(* CoDeSys 2.3.9.59 project: CIP_2k.pro *)
(* Author: Damir *)
(* Libraries: My_lib.lib 13.7.21 19:36:35, SysLibTime.lib 8.11.10 13:37:48, C:\Program Files (x86)\WAGO Software\CODESYS V2.3\Targets\WAGO\Libraries\IO_IPC\Util.lib 29.6.15 10:12:14, Standard.lib, SYSLIBCALLBACK.LIB *)

(* PLC configuration (modules and I/O channels)
0750-0455 4 AI 4-20mA s.e. [Type_8_4_Channels] node 0, in %IB32 out %QB8 {INTTypePAAssignment = PLC; INTTypeModule = plugged}
  AT %IW0 [WORDOnW_I] Ch_1 Input word
  AT %IW1 [WORDOnW_I] Ch_2 Input word
  AT %IW2 [WORDOnW_I] Ch_3 Input word
  AT %IW3 [WORDOnW_I] Ch_4 Input word
0750-0455 4 AI 4-20mA s.e. [Type_8_4_Channels] node 1, in %IB32 out %QB8 {INTTypePAAssignment = PLC; INTTypeModule = plugged}
  AT %IW4 [WORDOnW_I] Ch_1 Input word
  AT %IW5 [WORDOnW_I] Ch_2 Input word
  AT %IW6 [WORDOnW_I] Ch_3 Input word
  AT %IW7 [WORDOnW_I] Ch_4 Input word
0750-0455 4 AI 4-20mA s.e. [Type_8_4_Channels] node 2, in %IB40 out %QB8 {INTTypePAAssignment = PLC; INTTypeModule = plugged}
  AT %IW8 [WORDOnW_I] Ch_1 Input word
  AT %IW9 [WORDOnW_I] Ch_2 Input word
  AT %IW10 [WORDOnW_I] Ch_3 Input word
  AT %IW11 [WORDOnW_I] Ch_4 Input word
0750-0455 4 AI 4-20mA s.e. [Type_8_4_Channels] node 3, in %IB48 out %QB8 {INTTypePAAssignment = PLC; INTTypeModule = plugged}
  AT %IW12 [WORDOnW_I] Ch_1 Input word
  AT %IW13 [WORDOnW_I] Ch_2 Input word
  AT %IW14 [WORDOnW_I] Ch_3 Input word
  AT %IW15 [WORDOnW_I] Ch_4 Input word
0750-0555 4 AO 4-20mA [Type_14_4_Channels] node 8, in %IB56 out %QB8 {INTTypePAAssignment = PLC; INTTypeModule = plugged}
  AT %QW0 [WORDOnW_Q] Ch_1 Analog output
  AT %QW1 [WORDOnW_Q] Ch_2 Analog output
  AT %QW2 [WORDOnW_Q] Ch_3 Analog output
  AT %QW3 [WORDOnW_Q] Ch_4 Analog output
0750-0555 4 AO 4-20mA [Type_14_4_Channels] node 9, in %IB64 out %QB8 {INTTypePAAssignment = PLC; INTTypeModule = plugged}
  AT %QW4 [WORDOnW_Q] Ch_1 Analog output
  AT %QW5 [WORDOnW_Q] Ch_2 Analog output
  AT %QW6 [WORDOnW_Q] Ch_3 Analog output
  AT %QW7 [WORDOnW_Q] Ch_4 Analog output
0750-1405 16 DI 24V DC 3.0ms [Type_1_16_Channels] node 11, in %IB32 out %QB16 {INTTypePAAssignment = PLC; INTTypeModule = plugged}
  AT %IX16.0 [BOOLOnX_I] Ch_1 Digital input
  AT %IX16.1 [BOOLOnX_I] Ch_2 Digital input
  AT %IX16.2 [BOOLOnX_I] Ch_3 Digital input
  AT %IX16.3 [BOOLOnX_I] Ch_4 Digital input
  AT %IX16.4 [BOOLOnX_I] Ch_5 Digital input
  AT %IX16.5 [BOOLOnX_I] Ch_6 Digital input
  AT %IX16.6 [BOOLOnX_I] Ch_7 Digital input
  AT %IX16.7 [BOOLOnX_I] Ch_8 Digital input
  AT %IX16.8 [BOOLOnX_I] Ch_9 Digital input
  AT %IX16.9 [BOOLOnX_I] Ch_10 Digital input
  AT %IX16.10 [BOOLOnX_I] Ch_11 Digital input
  AT %IX16.11 [BOOLOnX_I] Ch_12 Digital input
  AT %IX16.12 [BOOLOnX_I] Ch_13 Digital input
  AT %IX16.13 [BOOLOnX_I] Ch_14 Digital input
  AT %IX16.14 [BOOLOnX_I] Ch_15 Digital input
  AT %IX16.15 [BOOLOnX_I] Ch_16 Digital input
0750-1405 16 DI 24V DC 3.0ms [Type_1_16_Channels] node 12, in %IB32 out %QB16 {INTTypePAAssignment = PLC; INTTypeModule = plugged}
  AT %IX17.0 [BOOLOnX_I] Ch_1 Digital input
  AT %IX17.1 [BOOLOnX_I] Ch_2 Digital input
  AT %IX17.2 [BOOLOnX_I] Ch_3 Digital input
  AT %IX17.3 [BOOLOnX_I] Ch_4 Digital input
  AT %IX17.4 [BOOLOnX_I] Ch_5 Digital input
  AT %IX17.5 [BOOLOnX_I] Ch_6 Digital input
  AT %IX17.6 [BOOLOnX_I] Ch_7 Digital input
  AT %IX17.7 [BOOLOnX_I] Ch_8 Digital input
  AT %IX17.8 [BOOLOnX_I] Ch_9 Digital input
  AT %IX17.9 [BOOLOnX_I] Ch_10 Digital input
  AT %IX17.10 [BOOLOnX_I] Ch_11 Digital input
  AT %IX17.11 [BOOLOnX_I] Ch_12 Digital input
  AT %IX17.12 [BOOLOnX_I] Ch_13 Digital input
  AT %IX17.13 [BOOLOnX_I] Ch_14 Digital input
  AT %IX17.14 [BOOLOnX_I] Ch_15 Digital input
  AT %IX17.15 [BOOLOnX_I] Ch_16 Digital input
0750-1405 16 DI 24V DC 3.0ms [Type_1_16_Channels] node 13, in %IB34 out %QB16 {INTTypePAAssignment = PLC; INTTypeModule = plugged}
  AT %IX18.0 [BOOLOnX_I] Ch_1 Digital input
  AT %IX18.1 [BOOLOnX_I] Ch_2 Digital input
  AT %IX18.2 [BOOLOnX_I] Ch_3 Digital input
  AT %IX18.3 [BOOLOnX_I] Ch_4 Digital input
  AT %IX18.4 [BOOLOnX_I] Ch_5 Digital input
  AT %IX18.5 [BOOLOnX_I] Ch_6 Digital input
  AT %IX18.6 [BOOLOnX_I] Ch_7 Digital input
  AT %IX18.7 [BOOLOnX_I] Ch_8 Digital input
  AT %IX18.8 [BOOLOnX_I] Ch_9 Digital input
  AT %IX18.9 [BOOLOnX_I] Ch_10 Digital input
  AT %IX18.10 [BOOLOnX_I] Ch_11 Digital input
  AT %IX18.11 [BOOLOnX_I] Ch_12 Digital input
  AT %IX18.12 [BOOLOnX_I] Ch_13 Digital input
  AT %IX18.13 [BOOLOnX_I] Ch_14 Digital input
  AT %IX18.14 [BOOLOnX_I] Ch_15 Digital input
  AT %IX18.15 [BOOLOnX_I] Ch_16 Digital input
0750-1504 16 DO 24V DC 0.5A [Type_10_16_Channels] node 19, in %IB36 out %QB16 {INTTypePAAssignment = PLC; INTTypeModule = plugged}
  AT %QX8.0 [BOOLOnX_Q] Ch_1 Digital output
  AT %QX8.1 [BOOLOnX_Q] Ch_2 Digital output
  AT %QX8.2 [BOOLOnX_Q] Ch_3 Digital output
  AT %QX8.3 [BOOLOnX_Q] Ch_4 Digital output
  AT %QX8.4 [BOOLOnX_Q] Ch_5 Digital output
  AT %QX8.5 [BOOLOnX_Q] Ch_6 Digital output
  AT %QX8.6 [BOOLOnX_Q] Ch_7 Digital output
  AT %QX8.7 [BOOLOnX_Q] Ch_8 Digital output
  AT %QX8.8 [BOOLOnX_Q] Ch_9 Digital output
  AT %QX8.9 [BOOLOnX_Q] Ch_10 Digital output
  AT %QX8.10 [BOOLOnX_Q] Ch_11 Digital output
  AT %QX8.11 [BOOLOnX_Q] Ch_12 Digital output
  AT %QX8.12 [BOOLOnX_Q] Ch_13 Digital output
  AT %QX8.13 [BOOLOnX_Q] Ch_14 Digital output
  AT %QX8.14 [BOOLOnX_Q] Ch_15 Digital output
  AT %QX8.15 [BOOLOnX_Q] Ch_16 Digital output
0750-1504 16 DO 24V DC 0.5A [Type_10_16_Channels] node 20, in %IB38 out %QB16 {INTTypePAAssignment = PLC; INTTypeModule = plugged}
  AT %QX9.0 [BOOLOnX_Q] Ch_1 Digital output
  AT %QX9.1 [BOOLOnX_Q] Ch_2 Digital output
  AT %QX9.2 [BOOLOnX_Q] Ch_3 Digital output
  AT %QX9.3 [BOOLOnX_Q] Ch_4 Digital output
  AT %QX9.4 [BOOLOnX_Q] Ch_5 Digital output
  AT %QX9.5 [BOOLOnX_Q] Ch_6 Digital output
  AT %QX9.6 [BOOLOnX_Q] Ch_7 Digital output
  AT %QX9.7 [BOOLOnX_Q] Ch_8 Digital output
  AT %QX9.8 [BOOLOnX_Q] Ch_9 Digital output
  AT %QX9.9 [BOOLOnX_Q] Ch_10 Digital output
  AT %QX9.10 [BOOLOnX_Q] Ch_11 Digital output
  AT %QX9.11 [BOOLOnX_Q] Ch_12 Digital output
  AT %QX9.12 [BOOLOnX_Q] Ch_13 Digital output
  AT %QX9.13 [BOOLOnX_Q] Ch_14 Digital output
  AT %QX9.14 [BOOLOnX_Q] Ch_15 Digital output
  AT %QX9.15 [BOOLOnX_Q] Ch_16 Digital output
0750-1504 16 DO 24V DC 0.5A [Type_10_16_Channels] node 21, in %IB38 out %QB18 {INTTypePAAssignment = PLC; INTTypeModule = plugged}
  AT %QX10.0 [BOOLOnX_Q] Ch_1 Digital output
  AT %QX10.1 [BOOLOnX_Q] Ch_2 Digital output
  AT %QX10.2 [BOOLOnX_Q] Ch_3 Digital output
  AT %QX10.3 [BOOLOnX_Q] Ch_4 Digital output
  AT %QX10.4 [BOOLOnX_Q] Ch_5 Digital output
  AT %QX10.5 [BOOLOnX_Q] Ch_6 Digital output
  AT %QX10.6 [BOOLOnX_Q] Ch_7 Digital output
  AT %QX10.7 [BOOLOnX_Q] Ch_8 Digital output
  AT %QX10.8 [BOOLOnX_Q] Ch_9 Digital output
  AT %QX10.9 [BOOLOnX_Q] Ch_10 Digital output
  AT %QX10.10 [BOOLOnX_Q] Ch_11 Digital output
  AT %QX10.11 [BOOLOnX_Q] Ch_12 Digital output
  AT %QX10.12 [BOOLOnX_Q] Ch_13 Digital output
  AT %QX10.13 [BOOLOnX_Q] Ch_14 Digital output
  AT %QX10.14 [BOOLOnX_Q] Ch_15 Digital output
  AT %QX10.15 [BOOLOnX_Q] Ch_16 Digital output
Fieldbus variables [FB_VARS] node 1, in %IB0 out %QB0
Flag variables [FLAG_VARS] node 2, in %IB0 out %QB0
Modbus-Master [MB_MASTER] node 3, in %IB0 out %QB0
*)

(* Global variable list: Alarms *)
VAR_GLOBAL

(*----------------аварии контура 1---------------------*)
	Alarm_VA541		AT %QX256.0	: BOOL;	(*аварии клапанов*)
	Alarm_VA401    		AT %QX256.1 	: BOOL;
	Alarm_VA201    		AT %QX256.2  	: BOOL;
	Alarm_VA301    		AT %QX256.3 	: BOOL;
	Alarm_VA41     		AT %QX256.4  	: BOOL;
	Alarm_VA11     		AT %QX256.5	: BOOL;
	Alarm_VA21     		AT %QX256.6  	: BOOL;
	Alarm_VA31     		AT %QX256.7 	: BOOL;
	Alarm_VA5	    		AT %QX256.8  	: BOOL;
	Alarm_VA501    		AT %QX256.9  	: BOOL;
	Alarm_VA51     		AT %QX256.10  	: BOOL;
	Alarm_VA511    		AT %QX256.11  	: BOOL;
	Alarm_VA521    		AT %QX256.12  	: BOOL;
	Alarm_VA531    		AT %QX256.13  	: BOOL;
	Alarm_P1       		AT %QX256.14  	: BOOL;	(*авария насоса подачи*)
	Alarm_PE1        		AT %QX256.15  	: BOOL;	(*Превышение давления контур 1*)

	Alarm_FE11      		AT %QX257.0	: BOOL;	(*Нет протока на подаче контур 1*)
	AlarmBackFlow_C1 	AT %QX257.1 	: BOOL; 	(*Нет протока на возврате контур 1*)
	HeatingAlarm_C1  	AT %QX257.2 	: BOOL; 	(*Долгий нагрев контур 1*)
	CondAlarm_C1  		AT %QX257.3 	: BOOL; 	(*Долгий набор концентрации контур 1*)
	Alarm_Empty_Q5		AT %QX257.4 	: BOOL; 	(*авария опустошения цирк бака при работе на замкн маршруте*)
	Alarm_TE11      		AT %QX257.5  	: BOOL; 	(*Перегрев на выходе теплообменника контура 1*)

	Error_TE11      	AT %QX258.0 	: BOOL; (*аварии аналоговых датчиков*)
	Error_PE1        	AT %QX258.1 	: BOOL;
	Error_FE1        	AT %QX258.2  	: BOOL;
	Error_QE1        	AT %QX258.3  	: BOOL;
	Error_TE21       	AT %QX258.4  	: BOOL;


(*-----------------аварии контура 2-------------------*)
	Alarm_VA642    	AT %QX259.0  	: BOOL;
	Alarm_VA402    	AT %QX259.1  	: BOOL;
	Alarm_VA202    	AT %QX259.2 	: BOOL;
	Alarm_VA302    	AT %QX259.3 	: BOOL;
	Alarm_VA42    	AT %QX259.4  	: BOOL;
	Alarm_VA12     	AT %QX259.5  	: BOOL;
	Alarm_VA22     	AT %QX259.6 	: BOOL;
	Alarm_VA32     	AT %QX259.7 	: BOOL;
	Alarm_VA6	    	AT %QX259.8  	: BOOL;
	Alarm_VA602    	AT %QX259.9  	: BOOL;
	Alarm_VA62     	AT %QX259.10  	: BOOL;
	Alarm_VA612    	AT %QX259.11 	: BOOL;
	Alarm_VA622    	AT %QX259.12 	: BOOL;
	Alarm_VA632    	AT %QX259.13 	: BOOL;
	Alarm_P2       	AT %QX259.14  	: BOOL;	(*авария насоса подачи*)
	Alarm_PE2        	AT %QX259.15  	: BOOL; 	(*Превышение давления контур 2*)

	Alarm_FE12       		AT %QX260.0  	: BOOL;	(*Нет протока на подаче контур 2*)
	AlarmBackFlow_C2 	AT %QX260.1	: BOOL; 	(*Нет протока на возврате контур 2*)
	HeatingAlarm_C2  	AT %QX260.2  	: BOOL; 	(*Долгий нагрев контур 2*)
	CondAlarm_C2  		AT %QX260.3 	: BOOL; 	(*Долгий набор концентрации контур 2*)
	Alarm_Empty_Q6   	AT %QX260.4 	: BOOL; 	(*авария опустошения цирк бака при работе на замкн маршруте*)
	Alarm_TE12      		AT %QX260.5  	: BOOL; 	(*Перегрев на выходе теплообменника контура 2*)

	Error_TE12       	AT %QX261.0  	: BOOL;	(*аварии аналоговых датчиков*)
	Error_PE2        	AT %QX261.1 	: BOOL;
	Error_FE2        	AT %QX261.2  	: BOOL;
	Error_QE2        	AT %QX261.3  	: BOOL;
	Error_TE22       	AT %QX261.4  	: BOOL;

(*-----------------аварии контура 3-------------------*)
(*%QX262 - %QX264*)


(*------------------общие аварии---------------------*)
	Alarm_PS         		AT %QX268.0  	: BOOL; 	(*Низкое давление сжатого воздуха*)
	Alarm_Stop       		AT %QX268.1  	: BOOL; 	(*Аварийный стоп*)
	Power_loss       		AT %QX268.2  	: BOOL; 	(*подача питания на плк - перезагрузка*)
	Alarm_VA1      		AT %QX268.3  	: BOOL;		(*авария клапана подачи чистой воды в танк Q1*)
	Alarm_LS81      		AT %QX268.4  	: BOOL;		(*аварийный уровень в баке концентрата кислоты*)
	Alarm_LS82      		AT %QX268.5  	: BOOL; 	(*низкий уровень в баке концентрата кислоты*)
	Alarm_LS71      		AT %QX268.6  	: BOOL; 	(*аварийный уровень в баке концентрата щелочи*)
	Alarm_LS72      		AT %QX268.7  	: BOOL; 	(*низкий уровень в баке концентрата щелочи*)
	Alarm_LS91     		AT %QX268.8  	: BOOL; 	(*аварийный уровень в баке дезинфектанта*)
	Alarm_LS92    		AT %QX268.9  	: BOOL; 	(*низкий уровень в баке дезинфектанта*)
    	Alarm_MinLev_Q1	AT %QX268.10  	: BOOL; 	(*минимальный уровень в танке чистой воды*)
    	Alarm_MinLev_Q2 	AT %QX268.11  	: BOOL; 	(*минимальный уровень в танке щелочи*)
    	Alarm_MinLev_Q3 	AT %QX268.12  	: BOOL; 	(*минимальный уровень в танке кислоты*)


	Error_TE2        	AT %QX269.0	: BOOL;	(*аварии аналоговых датчиков*)
	Error_TE3        	AT %QX269.1  	: BOOL;
	Error_LE1        	AT %QX269.2  	: BOOL;
	Error_LE2        	AT %QX269.3  	: BOOL;
	Error_LE3        	AT %QX269.4 	: BOOL;
(*	Error_LE4        	AT %QX269.5 	: BOOL;
	Error_TE4        	AT %QX269.6  	: BOOL; *)








END_VAR

(* Global variable list: AnalogScale *)
VAR_GLOBAL
(*%QX270 - %QX362*)

(*----------------масштабированные и пересчитанные  значения-----------------------*)
(*контур 1*)
	i_TE11   				AT %QW270		: REAL;		(*температура подачи контур 1*)
	QE1         				AT %QW272 	: REAL;     	(*расчитанная концентрация % раствора контур 1*)
	i_TE21      				AT %QW274 	: REAL;    	(*температура возврата контур 1*)
	i_FE1       				AT %QW276 	: REAL;    	(*производительность подачи л/час контур 1*)
	i_PE1       				AT %QW278 	: REAL;  	(*давление подачи контура 1*)
	i_QE1       				AT %QW280 	: REAL;  	(*показание концентратомера контур 1, мСм/см*)
	QE1_priv    				AT %QW282 	: REAL;     	(*приведенная проводимость к температуре контур 1*)
	Current_VolumeFC1		AT %QW284		: REAL;		(*текуший объем расходомера дезинфектанта контур 1*)
	Current_VolumeFC11		AT %QW286		: REAL;		(*текуший объем расходомера подачи контур 1*)

(*контур 2*)
	i_TE12      				AT %QW290 	: REAL;   	(*температура подачи контур 2*)
	QE2        				AT %QW292 	: REAL;     	(*расчитанная концентрация % раствора контур 2*)
	i_TE22      				AT %QW294 	: REAL;   	(*температура возврата контур 2*)
	i_FE2       				AT %QW296 	: REAL;   	(*производительность подачи л/час контур 2*)
	i_PE2       				AT %QW298 	: REAL;  	(*давление подачи контура 2*)
	i_QE2       				AT %QW300 	: REAL;  	(*показание концентратомера контур 2, мСм/см*)
	QE2_priv    				AT %QW302 	: REAL;     	(*приведенная проводимость к температуре контур 2*)
	Current_VolumeFC2     	AT %QW304		: REAL;  	(*текуший объем расходомера дезинфектанта контур 2*)
	Current_VolumeFC12 	AT %QW306		: REAL;		(*текуший объем расходомера подачи контур 2*)

(*контур 3*)
(*%QX310 - %QX326*)


(*общие*)
	i_TE2       	AT %QW340 	: REAL;  	(*температура в танке щелочи*)
	i_TE3       	AT %QW342 	: REAL;  	(*температура в танке кислоты*)
	i_LE1       	AT %QW344 	: REAL;   	(*текущий уровень в танке чистой воды %*)
	i_LE2       	AT %QW346 	: REAL;   	(*текущий уровень в танке щелочи %*)
	i_LE3       	AT %QW348 	: REAL;   	(*текущий уровень в танке кислоты %*)
(*	i_LE4       	AT %QW350 	: REAL;   	(*текущий уровень в танке возвратной воды %*)
	i_TE4       	AT %QW352 	: REAL;  	(*температура в танке возвратной воды*) *)


END_VAR

VAR_GLOBAL RETAIN
(*структуры данных для масштабирования сигналов с аналоговых датчиков, пользовательский тип данных AnalogScale *)
(*----------------------Контур 1----------------------------------*)
	An_Scale_TE11		AT %MW0	: AnalogScale:=(Zero:=FALSE, MaxKod:=32764.0, MinKod:=0.0, MaxVal:=100.0, MinVal:=0.0, ErrorLevel:=0.01, NumbSample:=200);
	An_Scale_PE1		AT %MW20	: AnalogScale:=(Zero:=FALSE, MaxKod:=32764.0, MinKod:=0.0, MaxVal:=6.0, MinVal:=0.0, ErrorLevel:=0.01, NumbSample:=200);
	An_Scale_FE1		AT %MW40	: AnalogScale:=(Zero:=FALSE, MaxKod:=32764.0, MinKod:=0.0, MaxVal:=30000.0, MinVal:=0.0, ErrorLevel:=0.01, NumbSample:=200);
	An_Scale_QE1		AT %MW60	: AnalogScale:=(Zero:=FALSE, MaxKod:=32764.0, MinKod:=0.0, MaxVal:=500.0, MinVal:=0.0, ErrorLevel:=0.01, NumbSample:=200);
	An_Scale_TE21		AT %MW80	: AnalogScale:=(Zero:=FALSE, MaxKod:=32764.0, MinKod:=0.0, MaxVal:=100.0, MinVal:=0.0, ErrorLevel:=0.01, NumbSample:=200);

(*----------------------Контур 2----------------------------------*)
	An_Scale_TE12		AT %MW100	: AnalogScale:=(Zero:=FALSE, MaxKod:=32764.0, MinKod:=0.0, MaxVal:=100.0, MinVal:=0.0, ErrorLevel:=0.01, NumbSample:=200);
	An_Scale_PE2		AT %MW120	: AnalogScale:=(Zero:=FALSE, MaxKod:=32764.0, MinKod:=0.0, MaxVal:=6.0, MinVal:=0.0, ErrorLevel:=0.01, NumbSample:=200);
	An_Scale_FE2		AT %MW140	: AnalogScale:=(Zero:=FALSE, MaxKod:=32764.0, MinKod:=0.0, MaxVal:=30000.0, MinVal:=0.0, ErrorLevel:=0.01, NumbSample:=200);
	An_Scale_QE2		AT %MW160	: AnalogScale:=(Zero:=FALSE, MaxKod:=32764.0, MinKod:=0.0, MaxVal:=500.0, MinVal:=0.0, ErrorLevel:=0.01, NumbSample:=200);
	An_Scale_TE22		AT %MW180	: AnalogScale:=(Zero:=FALSE, MaxKod:=32764.0, MinKod:=0.0, MaxVal:=100.0, MinVal:=0.0, ErrorLevel:=0.01, NumbSample:=200);

(*----------------------общие--------------------------------*)
	An_Scale_TE2		AT %MW200	: AnalogScale:=(Zero:=FALSE, MaxKod:=32764.0, MinKod:=0.0, MaxVal:=100.0, MinVal:=0.0, ErrorLevel:=0.01, NumbSample:=200);
	An_Scale_TE3		AT %MW220	: AnalogScale:=(Zero:=FALSE, MaxKod:=32764.0, MinKod:=0.0, MaxVal:=100.0, MinVal:=0.0, ErrorLevel:=0.01, NumbSample:=200);
	An_Scale_LE1		AT %MW240	: AnalogScale:=(Zero:=FALSE, MaxKod:=32764.0, MinKod:=0.0, MaxVal:=0.25, MinVal:=0.0, ErrorLevel:=0.01, Hight_LE:=2.4, NumbSample:=200);
	An_Scale_LE2		AT %MW260	: AnalogScale:=(Zero:=FALSE, MaxKod:=32764.0, MinKod:=0.0, MaxVal:=0.25, MinVal:=0.0, ErrorLevel:=0.01, Hight_LE:=2.4, NumbSample:=200);
	An_Scale_LE3		AT %MW280	: AnalogScale:=(Zero:=FALSE, MaxKod:=32764.0, MinKod:=0.0, MaxVal:=0.25, MinVal:=0.0, ErrorLevel:=0.01, Hight_LE:=2.4, NumbSample:=200);
(*	An_Scale_LE4		AT %MW300	: AnalogScale:=(Zero:=FALSE, MaxKod:=32764.0, MinKod:=0.0, MaxVal:=0.25, MinVal:=0.0, ErrorLevel:=0.01 ,Hight_LE:=2.4, NumbSample:=200);
	An_Scale_TE4		AT %MW320	: AnalogScale:=(Zero:=FALSE, MaxKod:=32764.0, MinKod:=0.0, MaxVal:=100.0, MinVal:=0.0, ErrorLevel:=0.01, NumbSample:=200); *)



END_VAR

(* Global variable list: Constants *)
VAR_GLOBAL CONSTANT

	ar_Null_20 : ARRAY [0..20] OF BOOL := 21(FALSE) ;  (*нулевой массив для обнуления*)
	ar_Full_20 : ARRAY [0..20] OF BOOL := 21(TRUE) ;    (*заполненный массив*)

(*объявления констант для доступа к отдельным битам в словах *)
(*управление механизмами каждого контура*)
	VA541		: INT:= 0;	(*VA541 Клапан сброса в канализацию из контура *)
	VA401		: INT:= 1;	(*VA401 Клапан подачи в бак возвратной воды *)
	VA201		: INT:= 2;	(*VA201 Клапан подачи в бак щелочи *)
	VA301		: INT:= 3;	(*VA301 Клапан подачи в бак кислоты *)
	VA41		: INT:= 4;	(*VA41 Клапан выпуска из бака возвратной воды*)
	VA11		: INT:= 5;	(*VA11 Клапан выпуска из бака чистой воды*)
	VA21		: INT:= 6;	(*VA21 Клапан выпуска из бака щелочи*)
	VA31		: INT:= 7;	(*VA31 Клапан выпуска из бака кислоты*)
	VA5			: INT:= 8;	(*VA5 Клапан подачи чистой воды в цирк бак*)
	VA501		: INT:= 9;	(*VA501 Клапан подачи растворов в цирк бак*)
	VA51		: INT:= 10;	(*VA51  Клапан выпуска из цирк бака*)
	VA511		: INT:= 11;	(*VA511 Клапан выпуска в канализацию из цирк бака*)
	VA521		: INT:= 12;	(*VA521 Клапан циркуляции по контуру*)
	VA531		: INT:= 13;	(*VA531 Клапан подачи из контура в маршрут*)
	VA14		: INT:= 14;	(*VA14 Отсечной клапан пара*)
	P1			: INT:= 15;	(*Р1 Старт насоса подачи *)

	BackPump		: INT:= 16;	(*Старт насоса возврата*)
	Heating_VR1		: INT:= 17;	(*Включение нагрева*)
	VE551			: INT:= 18;	(*VE551 Клапан дезинфектанта*)
	Zero_FC11		: INT:= 19;	(*обнуление счетчика расходомера раствора, в ручном режиме*)
	Zero_FC1		: INT:= 20;	(*обнуление счетчика расходомера дезинфектанта, в ручном режиме*)


END_VAR

(* Global variable list: DeviceControl *)
VAR_GLOBAL

(*-------------состояние механизмов с диагностикой контур 1-------------*)
	Mode_VA541 	AT %QW360: INT;
	Mode_VA401    	AT %QW361: INT;
	Mode_VA201    	AT %QW362: INT;
	Mode_VA301    	AT %QW363: INT;
	Mode_VA41     	AT %QW364: INT;
	Mode_VA11     	AT %QW365: INT;
	Mode_VA21     	AT %QW366: INT;
	Mode_VA31     	AT %QW367: INT;
	Mode_VA5    	AT %QW368: INT;
	Mode_VA501    	AT %QW369: INT;
	Mode_VA51     	AT %QW370: INT;
	Mode_VA511    	AT %QW371: INT;
	Mode_VA521    	AT %QW372: INT;
	Mode_VA531    	AT %QW373: INT;
	Mode_P1     		AT %QW374: INT;


(*-------------состояние  механизмов с диагностикой контур 2-------------*)
	Mode_VA642    	AT %QW380: INT;
	Mode_VA402    	AT %QW381: INT;
	Mode_VA202    	AT %QW382: INT;
	Mode_VA302    	AT %QW383: INT;
	Mode_VA42    	AT %QW384: INT;
	Mode_VA12     	AT %QW385: INT;
	Mode_VA22     	AT %QW386: INT;
	Mode_VA32     	AT %QW387: INT;
	Mode_VA6    	AT %QW388: INT;
	Mode_VA602    	AT %QW389: INT;
	Mode_VA62     	AT %QW390: INT;
	Mode_VA612    	AT %QW391: INT;
	Mode_VA622    	AT %QW392: INT;
	Mode_VA632    	AT %QW393: INT;
	Mode_P2     		AT %QW394: INT;

(*-------------состояние механизмов с диагностикой контур 3-------------*)
(*%QW400 - %QW414*)


(*------------состояние общих механизмов с диагностикой--------------*)
	Mode_VA1      	AT %QW439: INT;

(*------------------------------------------------------------------------------------------*)

(*------------------команды управления механизмами------------------*)
(*контур 1*)
	w_qDevice_C1		AT%QW440	:DWORD; 	(*слово команд управления механизмами контура 1*)
	q_P1an  			AT%QW442 	: REAL;		(*аналоговое задание на насос подачи*)
	q_VR1an 			AT%QW444 	: REAL;		(*аналоговое задание на регулирующий клапан пара*)
	SP_VR1							: REAL;		(*задание температуры на регулятор*)
	SP_P1  							: REAL;	 	(*задание производительности на регулятор*)

(*контур 2*)
	w_qDevice_C2		AT%QW446	:DWORD; 	(*слово команд управления механизмами контура 2*)
	q_P2an  			AT%QW448 	: REAL;
	q_VR2an 			AT%QW450 	: REAL;
	SP_VR2 						: REAL;	 	(*задание температуры на регулятор*)
	SP_P2  							: REAL;	 	(*задание производительности на регулятор*)

(*контур 3*)
(*%QW452 - %QW458*)

(*общие механизмы*)
	q_VA1      			AT %QX462.0	: BOOL;		(*VA1  Клапан подачи в бак чистой воды*)
	q_VE7     			AT %QX462.1	: BOOL;		(*VE7 Клапан промывки линии концентрата щелочи*)
	q_P8     				AT %QX462.2	: BOOL;		(*Р8 Насос-дозатор концентрата  кислоты*)
	q_P9     				AT %QX462.3	: BOOL;		(*Р9 Насос-дозатор концентрата  щелочи*)
	q_P10     			AT %QX462.4	: BOOL;		(*Р10 Насос-дозатор дезинфектанта*)

(*----------------------------------------------------------------------------------*)





END_VAR

VAR_GLOBAL RETAIN
(*вкл/выкл контроля положения клапанов*)
	wDiagVA_C1		AT%MW400		:WORD:= 16#FF ;	(*контроль состояния клапанов с диагностикой контур 1*)
	wDiagVA_C2		AT%MW401		:WORD:= 16#FF;	(*контроль состояния клапанов с диагностикой контур 2*)
	DiagVA1      			AT %MX402.0  	: BOOL:= TRUE;		(*контроль состояния клапана подачи в танк чистой воды*)

(*--------настройки ПИД-регуляторов-------------*)
(*контур 1*)
	SP_PID_P_VR1		AT %MW404	: REAL := 1.3;     	(*коеф усиления ПИД р-ра температуры*)
	SP_PID_I_VR1   	AT %MW406	: REAL := 10.0;    	(*время интегрирования ПИД р-ра температуры *)
	SP_PID_P_P1    	AT %MW408	: REAL := 0.5;     	(*коеф усиления ПИД р-ра расхода*)
	SP_PID_I_P1     		AT %MW410	: REAL := 10.0;    	(*время интегрирования ПИД р-ра расхода *)

(*контур 2*)
	SP_PID_P_VR2		AT %MW412	: REAL := 1.3;     	(*коеф усиления ПИД р-ра температуры*)
	SP_PID_I_VR2 		AT %MW414	: REAL := 10.0; 		(*время интегрирования ПИД р-ра температуры *)
	SP_PID_P_P2   		AT %MW416	: REAL := 0.3;     	(*коеф усиления ПИД р-ра расхода*)
	SP_PID_I_P2    		AT %MW418	: REAL := 10.0;    	(*время интегрирования ПИД р-ра расхода *)

(*------------вес импульса расходомера--------------*)
(*контур 1*)
	K_imp_C1         		AT %MW438	: REAL := 0.1;    		(*литр/имп расходомера подачи*)
	K_imp_dez_C1 		AT %MW440	: REAL := 5.0;     	(*мл/имп расходомера дезинфектанта*)
(*контур 2*)
	K_imp_C2        		AT %MW442	: REAL := 0.1;		(*литр/имп расходомера подачи*)
	K_imp_dez_C2 		AT %MW444	: REAL := 5.0;		(*мл/имп расходомера дезинфектанта*)


END_VAR

(* Global variable list: Global_Variables *)
VAR_GLOBAL
	scan_time : REAL;    (*время скана, из fb_TimeIncr*)


END_VAR

VAR_GLOBAL RETAIN

	Mode_Q1               	AT %MW500	: INT;  		(*режим пополнения бака Q1 чистой воды*)
	MaxLevel_Q1           	AT %MW501	: INT := 90;	(*макс уровень в танке чистой воды - поддержание уровня,%*)
	MinLevel_Q1          	AT %MW502	: INT := 70;  	(*мин уровень в танке чистой воды - поддержание уровня,%*)

	MinAlarmLevel_Q1   	AT %MW503	: INT := 20; 	(*мин уровень в танке чистой воды Q1,%*)
	MinAlarmLevel_Q2   	AT %MW504	: INT := 20;  	(*мин уровень в танке щелочи Q2,%*)
	MinAlarmLevel_Q3  	AT %MW505	: INT := 20;  	(*мин уровень в танке кислоты Q3,%*)
	MinAlarmLevel_Q4  	AT %MW506	: INT := 20;  	(*мин уровень в танке возврат воды Q4,%*)

	Time_LSH_on          	AT %MW508	: DINT := 1;		(*время задержки датчика верхнего уровня в цирк баке,сек*)
	Time_LSM_on         	AT %MW510	: DINT := 3; 		(*время задержки датчика среднего уровня в цирк баке,сек*)
	Time_LSM_off       	AT %MW512	: DINT := 2; 		(*время задержки датчика среднего уровня в цирк баке,сек*)
	Time_LSL_off       	AT %MW514	: DINT := 2; 		(*время задержки датчика нижнего уровня в цирк баке,сек*)

	Time_Control_TE    	AT %MW516	: DINT := 7; 		(*контрольное время набора температуры, мин*)
	Time_Control_QE    	AT %MW518	: DINT := 10;		(*контрольное время набора концентрации, мин*)
	Time_Alarm_FE       	AT %MW520	: DINT := 18;		(*время аварии протока на подаче, сек*)

	MaxPressure_C1   	AT %MW524	: REAL := 4.3;     (*уставка аварии по давлению контур 1*)
	MaxPressure_C2    	AT %MW526	: REAL := 4.3;     (*уставка аварии по давлению контур 2*)

	TimeDelay_C1       	AT %MW528	: DINT := 2;       	(*время задержки вкл/выкл клапанов и насосов контур 1*)
	TimeDelay_C2      	AT %MW530	: DINT := 2;       	(*время задержки вкл/выкл клапанов и насосов контур 2*)








END_VAR

(* Global variable list: HandMode *)
VAR_GLOBAL

    (*контур 1*)
	w_ManDevice_C1	AT%MW600	:DWORD; 	(*слово команд ручного режима контура 1*)
	ManSP_P1        		AT%MW602 : REAL;		(*задание производительности насоса подачи в ручном режиме*)
	ManSP_VR1       	AT%MW604 : REAL;		(*задание температуры нагрева в ручном режиме*)


    (*контур 2*)
	w_ManDevice_C2	AT%MW606	:DWORD; 	(*слово команд ручного режима контура 2*)
	ManSP_P2        		AT%MW608 : REAL;		(*задание производительности насоса подачи в ручном режиме*)
	ManSP_VR2       	AT%MW610 : REAL;		(*задание температуры нагрева в ручном режиме*)


    (*общие механизмы*)
	Man_VA1        	AT %MX626.0 	: BOOL;		(*VA1  Клапан подачи в бак чистой воды*)
	Man_VE7        	AT %MX626.1 	: BOOL;		(*VE7 Клапан промывки линии концентрата щелочи*)
	Man_P8          	AT %MX626.2 	: BOOL;		(*Р8 Насос-дозатор концентрата  кислоты*)
	Man_P9         	AT %MX626.3	: BOOL;		(*Р9 Насос-дозатор концентрата  щелочи*)
	Man_P10         	AT %MX626.4	: BOOL;		(*Р10 Насос-дозатор дезинфектанта*)

END_VAR

(* Global variable list: Inputs *)
VAR_GLOBAL
(*---------------переменные привязанные к физическим входам----------------------------*)

(*аналоговые входа*)
	TE11_i 	AT %IW0:  WORD;	(*ТЕ11 Температура на выходе нагревателя контур 1*)
	TE12_i 	AT %IW1:  WORD;	(*ТЕ12 Температура на выходе нагревателя контур 2*)
	TE2_i   	AT %IW2:  WORD;	(*ТЕ2 Температура в танке раствора щелочи Q2*)
	TE3_i	AT %IW3:  WORD;	(*ТЕ3 Температура в танке раствора кислоты Q3*)

	LE1_i  	AT %IW4:  WORD;	(*LE1 Датчик уровня в баке чистой воды*)
	LE2_i  	AT %IW5:  WORD;	(*LE2 Датчик уровня в баке щелочи*)
	LE3_i  	AT %IW6:  WORD;	(*LE3 Датчик уровня в баке кислоты*)
	PE1_i  	AT %IW7:  WORD;	(*PE1 Датчик давления контур 1*)

	PE2_i  	AT %IW8:  WORD;	(*PE2 Датчик давления контур 2*)
	FE1_i  	AT %IW9:  WORD;	(*Производительность подачи контур 1*)
	FE2_i 	AT %IW10: WORD;	(*Производительность подачи контур 2*)
(*	    		AT %IW11: WORD;	резерв*)

	QE1_i  	AT %IW12: WORD;	(*QE1 Проводимость контур 1*)
	TE21_i 	AT %IW13: WORD;	(*TE21 Температура на возврате контур 1*)
	QE2_i   	AT %IW14: WORD;	(*QE2 Проводимость контур 2*)
	TE22_i 	AT %IW15: WORD;	(*TE22 Температура на возврате контур 2*)

(*дискретные входа*)
	VA541_i		AT %IX16.0:  BOOL; 	(*датчик положения клапана*)
	VA642_i   	AT %IX16.1:  BOOL;	(*датчик положения клапана*)
	VA401_i    	AT %IX16.2:  BOOL;	(*датчик положения клапана*)
	VA402_i    	AT %IX16.3:  BOOL;	(*датчик положения клапана*)
	VA1_i         	AT %IX16.4:  BOOL;	(*датчик положения клапана*)
	VA201_i      	AT %IX16.5:  BOOL;	(*датчик положения клапана*)
	VA202_i      	AT %IX16.6:  BOOL;	(*датчик положения клапана*)
	VA301_i     	AT %IX16.7:  BOOL;	(*датчик положения клапана*)
	VA302_i     	AT %IX16.8:  BOOL;	(*датчик положения клапана*)
	VA41_i     	AT %IX16.9:  BOOL;	(*датчик положения клапана*)
	VA42_i      	AT %IX16.10: BOOL;	(*датчик положения клапана*)
	VA11_i      	AT %IX16.11: BOOL;	(*датчик положения клапана*)
	VA12_i     	AT %IX16.12: BOOL;	(*датчик положения клапана*)
	VA21_i     	AT %IX16.13: BOOL;	(*датчик положения клапана*)
	VA22_i     	AT %IX16.14: BOOL;	(*датчик положения клапана*)
	VA31_i     	AT %IX16.15: BOOL;	(*датчик положения клапана*)

	VA32_i      	AT %IX17.0:  BOOL;	(*датчик положения клапана*)
	VA5_i       	AT %IX17.1:  BOOL;	(*датчик положения клапана*)
	VA501_i      	AT %IX17.2:  BOOL;	(*датчик положения клапана*)
	VA51_i     	AT %IX17.3:  BOOL;	(*датчик положения клапана*)
	VA511_i      	AT %IX17.4:  BOOL;	(*датчик положения клапана*)
	FS21_i      	AT %IX17.5:  BOOL;	(*FS21 Датчик протока на возврате контура 1*)
	VA521_i     	AT %IX17.6:  BOOL;	(*датчик положения клапана*)
	VA531_i     	AT %IX17.7:  BOOL;	(*датчик положения клапана*)
	LSL5_i      	AT %IX17.8:  BOOL;	(*LSL5 Датчик нижнего уровня в цирк баке Q5*)
	LSM5_i     	AT %IX17.9:  BOOL;	(*LSM5 Датчик среднего уровня в цирк баке Q5*)
	LSH5_i      	AT %IX17.10: BOOL;	(*LSH5 Датчик верхнего уровня в цирк баке Q5*)
	VA6_i        	AT %IX17.11: BOOL;	(*датчик положения клапана*)
	VA602_i   	AT %IX17.12: BOOL;	(*датчик положения клапана*)
	VA62_i       	AT %IX17.13: BOOL;	(*датчик положения клапана*)
	VA612_i      	AT %IX17.14: BOOL;	(*датчик положения клапана*)
	FS22_i      	AT %IX17.15: BOOL;	(*FS22 Датчик протока на возврате контура 2*)


	VA622_i      	AT %IX18.0:  BOOL;	(*датчик положения клапана*)
	VA632_i      	AT %IX18.1:  BOOL;	(*датчик положения клапана*)
	LSL6_i       	AT %IX18.2:  BOOL;	(*LSL6 Датчик нижнего уровня в цирк баке Q6*)
	LSM6_i       	AT %IX18.3:  BOOL;	(*LSM6 Датчик среднего уровня в цирк баке Q6*)
	LSH6_i      	AT %IX18.4:  BOOL;	(*LSH6 Датчик верхнего уровня в цирк баке Q6*)
	LS71_i    	AT %IX18.5:  BOOL;	(*LS71 Датчик аварийного нижнего уровня в баке концентрата щелочи Q7*)
	LS72_i       	AT %IX18.6:  BOOL;	(*LS72 Датчик нижнего уровня в баке концентрата щелочи Q7*)
	LS81_i      	AT %IX18.7:  BOOL;	(*LS81 Датчик аварийного нижнего уровня в баке концентрата кислоты Q8*)
	LS82_i      	AT %IX18.8:  BOOL;	(*LS82 Датчик нижнего уровня в баке концентрата кислоты Q8*)
	PS1_i      	AT %IX18.9:  BOOL;	(*PS1 Датчик давления сжатого воздуха*)
	FC1_i       	AT %IX18.10: BOOL;	(*Расход раствора контур 1, имп*)
	FC2_i       	AT %IX18.11: BOOL;	(*Расход раствора контур 2, имп*)
	ProtectP1_i 	AT %IX18.12: BOOL;	(*Готовность частоного преобразователя насоса М1*)
	ProtectP2_i 	AT %IX18.13: BOOL;	(*Готовность частоного преобразователя насоса М2*)
	AlarmStop_i	AT %IX18.14: BOOL;	(*SB1 Аварийная стоповая кнопка пульта управления*)
(*	       		AT %IX18.15: BOOL;  резерв*)




END_VAR

(* Global variable list: OP_Comands *)
VAR_GLOBAL

	AlarmReset      					AT %MX700.0: BOOL; 	(*Сброс ошибок*)

END_VAR

(* Global variable list: Outputs *)
VAR_GLOBAL
(*переменные привязанные к физическим выходам*)
(*аналоговые выходы*)
	VR1an_q   	AT %QW0 : WORD;		(*VR1 Регулирующий клапан пара контур 1*)
	VR2an_q   	AT %QW1 : WORD;		(*VR2 Регулирующий клапан пара контур 2*)
(*   				AT %QW2 : WORD;
			   	AT %QW3 : WORD;  *)

	P1an_q    	AT %QW4 : WORD;		(*Задание скорости насоса подачи контура 1*)
	P2an_q    	AT %QW5 : WORD;		(*Задание скорости насоса подачи контура 2*)
(*			    	AT %QW6 : WORD;
			    	AT %QW7 : WORD;  *)


(*дискретные выходы*)
	q_Red    	AT %QX8.0  	: BOOL;		(*Светозвуковая сигнализация. Красный свет*)
	q_Yellow   	AT %QX8.1  	: BOOL;		(*Светозвуковая сигнализация. Желтый свет*)
	q_Green   	AT %QX8.2  	: BOOL;		(*Светозвуковая сигнализация. Зеленый свет*)
	q_Sirena   	AT %QX8.3  	: BOOL;		(*Светозвуковая сигнализация. Зуммер*)
	VE7_q   	AT %QX8.4  	: BOOL;		(*VE7 Клапан промывки линии концентрата щелочи*)
	P1_q     	AT %QX8.5  	: BOOL;		(*Старт частотного преобразователя насоса М1 контура 1*)
	P2_q   		AT %QX8.6  	: BOOL;		(*Старт частотного преобразователя насоса М2 контура 2*)
	H1_q   		AT %QX8.7  	: BOOL;		(*Насос возврата Н1*)
	H2_q   		AT %QX8.8  	: BOOL;		(*Насос возврата Н2*)
	H3_q   		AT %QX8.9  	: BOOL;		(*Насос возврата Н3*)
	H4_q   		AT %QX8.10	: BOOL;		(*Насос возврата Н4*)
	H5_q   		AT %QX8.11	: BOOL;		(*Насос возврата Н5*)
	H6_q   		AT %QX8.12	: BOOL;		(*Насос возврата Н6*)
	H7_q   		AT %QX8.13	: BOOL;		(*Насос возврата Н7*)
	H8_q   		AT %QX8.14	: BOOL;		(*Насос возврата Н8*)
	H9_q   		AT %QX8.15	: BOOL;		(*Насос возврата Н9*)

	VA541_q   	AT %QX9.0  	: BOOL;		(*VA541 Клапан сброса в канализацию из контура 1*)
	VA642_q   	AT %QX9.1  	: BOOL;		(*VA642 Клапан сброса в канализацию из контура 2*)
	VA1_q    	AT %QX9.2  	: BOOL;		(*VA1  Клапан подачи в бак чистой воды*)
	VA201_q    	AT %QX9.3  	: BOOL;		(*VA201 Клапан подачи в бак щелочи контур 1*)
	VA202_q    	AT %QX9.4  	: BOOL;		(*VA202 Клапан подачи в бак щелочи контур 2*)
	VA301_q    	AT %QX9.5  	: BOOL;		(*VA301 Клапан подачи в бак кислоты контур 1*)
	VA302_q    	AT %QX9.6  	: BOOL;		(*VA302 Клапан подачи в бак кислоты контур 2*)
	VA11_q    	AT %QX9.7  	: BOOL;		(*VA11 Клапан выпуска из бака чистой воды контур 1*)
	VA12_q    	AT %QX9.8  	: BOOL;		(*VA12 Клапан выпуска из бака чистой воды контур 2*)
	VA21_q    	AT %QX9.9  	: BOOL;		(*VA21 Клапан выпуска из бака щелочи контур 1*)
	VA22_q    	AT %QX9.10	: BOOL;		(*VA22 Клапан выпуска из бака щелочи контур 2*)
	VA31_q    	AT %QX9.11	: BOOL;		(*VA31 Клапан выпуска из бака кислоты контур 1*)
	VA32_q    	AT %QX9.12	: BOOL;		(*VA32 Клапан выпуска из бака кислоты контур 2*)
	VA5_q    	AT %QX9.13	: BOOL;		(*VA5 Клапан подачи чистой воды в цирк бак контур 1*)
	VA501_q    	AT %QX9.14	: BOOL;		(*VA501 Клапан подачи растворов в цирк бак контур 1*)
	VA51_q    	AT %QX9.15	: BOOL;		(*VA51  Клапан выпуска из цирк бака контур 1*)

	VA511_q    	AT %QX10.0	: BOOL;		(*VA511 Клапан выпуска в канализацию из цирк бака контур 1*)
	VA521_q    	AT %QX10.1	: BOOL;		(*VA521 Клапан циркуляции по контуру 1*)
	VA531_q   	AT %QX10.2	: BOOL;		(*VA531 Клапан подачи из контура 1*)
	VA14_q   	AT %QX10.3	: BOOL;		(*VA14 Отсечной клапан пара контур 1*)
	VA6_q    	AT %QX10.4	: BOOL;		(*VA6 Клапан подачи чистой воды в цирк бак контур 2*)
	VA602_q   	AT %QX10.5	: BOOL;		(*VA602 Клапан подачи растворов в цирк бак контур 2*)
	VA62_q   	AT %QX10.6	: BOOL;		(*VA62  Клапан выпуска из цирк бака контур 2*)
	VA612_q   	AT %QX10.7	: BOOL;		(*VA612 Клапан выпуска в канализацию из цирк бака контур 2*)
	VA622_q    	AT %QX10.8	: BOOL;		(*VA622 Клапан циркуляции по контуру 2*)
	VA632_q   	AT %QX10.9	: BOOL;		(*VA632 Клапан подачи из контура 2*)
	VA24_q   	AT %QX10.10: BOOL;			(*VA24 Отсечной клапан пара контур 2*)
	P8_q    		AT %QX10.11: BOOL;			(*Р8 Насос-дозатор концентрата  кислоты*)
	P9_q   		AT %QX10.12: BOOL;			(*Р9 Насос-дозатор концентрата  щелочи*)
(*	   			AT %QX10.13: BOOL;
	   			AT %QX10.14: BOOL;
	    			AT %QX10.15: BOOL; *)

END_VAR

(* Global variable list: Process_Settings *)
VAR_GLOBAL RETAIN

(*----------Контур 1---------------------*)
	AlkMixing_C1           			AT %MX800.0: BOOL;     		(*перемешивание щелочи*)
	AcidMixing_C1          			AT %MX800.1: BOOL;          	(*перемешивание кислоты*)

	Stop_C1                     		AT %MX801.0 : BOOL; 		(*принудительная остановка процесса*)
	Start_AutoWashing_C1        	AT %MX801.1 : BOOL; 		(*старт мойки в автомате*)
	Start_HandMode_C1           	AT %MX801.2 : BOOL; 		(*старт ручного режима*)
	Start_PrepareAlkaline_C1   	AT %MX801.3 : BOOL; 		(*старт подготовки раствора щелочи*)
	Start_PrepareAcid_C1        	AT %MX801.4 : BOOL; 		(*старт подготовки раствора кислоты*)
	Start_Diagnostic_C1         	AT %MX801.5 : BOOL; 		(*старт диагностики клапанов*)
	ch_SwillBackWater_C1        	AT %MX801.6 : BOOL:= FALSE; 		(*выбор операции мойки*)
	ch_SwillFreshWater_C1       	AT %MX801.7 : BOOL; 		(*выбор операции мойки*)
	ch_WashAlkaline_C1          	AT %MX801.8 : BOOL; 		(*выбор операции мойки*)
	ch_WashWater1_C1            	AT %MX801.9 : BOOL; 		(*выбор операции мойки*)
	ch_WashAcid_C1              	AT %MX801.10: BOOL;		(*выбор операции мойки*)
	ch_WashWater2_C1            	AT %MX801.11: BOOL; 		(*выбор операции мойки*)
	ch_ThermDesinfection_C1 	AT %MX801.12: BOOL; 		(*выбор операции мойки*)
	ch_ChemicDesinfection_C1	AT %MX801.13: BOOL:= FALSE; 		(*выбор операции мойки*)
	Pause_C1                    		AT %MX801.14: BOOL; 		(*пауза процесса*)


	TimeSwillBackWater_C1  		AT %MW810: DINT := 300;    	(*время полоскания возвратной водой,с*)
	TimeSwillFreshWater_C1 		AT %MW812: DINT := 300;   	(*время полоскания свежей водой,с*)
	TimeWashWater1_C1      		AT %MW814: DINT := 4;       	(*время мойки 1 чистой водой,мин*)
	TempWashWater1_C1      	AT %MW816: REAL := 40.0;  	(*температруа мойки 1 чистой водой*)
	TimeWashWater2_C1      		AT %MW818: DINT := 5;       	(*время мойки 2 чистой водой,мин*)
	TempWashWater2_C1      	AT %MW820: REAL := 40.0;  	(*температруа мойки 2 чистой водой*)
	TimeWashAlkaline_C1    		AT %MW822: DINT := 20;    	(*время мойки щелочью,мин*)
	TempWashAlkaline_C1    		AT %MW824: REAL := 75.0;  	(*температура мойки щелочью*)
	TimeAlkalineMix_C1     		AT %MW826: DINT := 60;     	(*время перемешивания при мойке щелочью,с*)
	TimeWashAcid_C1        		AT %MW828: DINT := 20;     	(*время мойки кислотой,мин*)
	TempWashAcid_C1        		AT %MW830: REAL := 65.0;  	(*температура мойки кислотой*)
	TimeAcidMix_C1         		AT %MW832: DINT := 60;     	(*время перемешивания при мойке кислотой,c*)
	TimeThermDesinf_C1     		AT %MW834: DINT := 10;     	(*время термической дезинфекции,мин*)
	TempThermDesinf_C1     		AT %MW836: REAL := 85.0;  	(*температура термической дезинфекции*)
	TempCoolThermDesinf_C1 	AT %MW838: REAL := 15.0;  	(*температура охлаждения терм дезинфекции*)
	TimeChemicDesinf_C1    		AT %MW840: DINT := 10;     	(*время химической дезинфекции,мин*)
	TimeSwillChemic_C1     		AT %MW842: DINT := 15;   	(*время ополаскивания чистой водой после хим дезинфекции*)
	TimeSwillWashWater1_C1    	AT %MW844: DINT := 5;  	(*время промывки водой со сбросом в Q4 после мойки 1 чистой водой,мин*)
	TimeSwillWashWater2_C1    	AT %MW846: DINT := 5;  	(*время промывки водой со сбросом в Q4 после мойки 2 чистой водой,мин*)

	(*рецепт*)
	RouteType_C1           		AT %MW870: DINT ;           	(*тип маршрута 1 - емкостной, 0 - замкнутый*)
	PumpCapacity_C1        		AT %MW872: DINT ;           	(*производительность подающего насоса *)
	TimeDelayRetPump_C1    	AT %MW874: DINT ;           	(*время задержки включения насоса возврата*)
	TimeDelayRetFlow_C1    		AT %MW876: DINT ;           	(*время появления протока на возврате*)
	TimeAlarmBackFlow_C1   		AT %MW878: DINT ;           	(*время аварии отсутствия обратного протока*)
	Numb_BackPump_C1       	AT %MW880: DINT ;           	(*номер насоса возврата*)
	VolumeDesinf_C1        		AT %MW882: DINT ;           	(*объем дезинфектанта*)
	Using_Q5_C1             		AT %MW884: DINT ;           	(*использование циркуляционного бака на мойках растворами и водой, 1 - использовать*)
	DeltaTempStartTime_C1  		AT %MW886: DINT ;           	(*перепад температуры TE1-TE2 для начала терм дезинфекции*)
	Route_C1               			AT %MW888: DINT ;           	(*номер выбранного маршрут контура*)


(*----------Контур 2---------------------*)
	AlkMixing_C2           			AT %MX900.0: BOOL;         	(*перемешивание щелочи*)
	AcidMixing_C2          			AT %MX900.1: BOOL;          	(*перемешивание кислоты*)

	Stop_C2                     		AT %MX901.0 : BOOL; 		(*принудительная остановка процесса*)
	Start_AutoWashing_C2        	AT %MX901.1 : BOOL; 		(*старт мойки в автомате*)
	Start_HandMode_C2           	AT %MX901.2 : BOOL; 		(*старт ручного режима*)
	Start_PrepareAlkaline_C2   	AT %MX901.3 : BOOL; 		(*старт подготовки раствора щелочи*)
	Start_PrepareAcid_C2        	AT %MX901.4 : BOOL; 		(*старт подготовки раствора кислоты*)
	Start_Diagnostic_C2         	AT %MX901.5 : BOOL; 		(*старт диагностики клапанов*)
	ch_SwillBackWater_C2        	AT %MX901.6 : BOOL:= FALSE; 		(*выбор операции мойки*)
	ch_SwillFreshWater_C2       	AT %MX901.7 : BOOL; 		(*выбор операции мойки*)
	ch_WashAlkaline_C2          	AT %MX901.8 : BOOL; 		(*выбор операции мойки*)
	ch_WashWater1_C2            	AT %MX901.9 : BOOL; 		(*выбор операции мойки*)
	ch_WashAcid_C2              	AT %MX901.10 : BOOL;		(*выбор операции мойки*)
	ch_WashWater2_C2            	AT %MX901.11: BOOL; 		(*выбор операции мойки*)
	ch_ThermDesinfection_C2  	AT %MX901.12: BOOL; 		(*выбор операции мойки*)
	ch_ChemicDesinfection_C2  	AT %MX901.13: BOOL:= FALSE; 		(*выбор операции мойки*)
	Pause_C2                    		AT %MX901.14: BOOL; 		(*пауза процесса*)


	TimeSwillBackWater_C2  		AT %MW910: DINT := 300;    	(*время полоскания возвратной водой,с*)
	TimeSwillFreshWater_C2 		AT %MW912: DINT := 300;    	(*время полоскания свежей водой,с*)
	TimeWashWater1_C2      		AT %MW914: DINT := 4;       	(*время мойки 1 чистой водой,мин*)
	TempWashWater1_C2      	AT %MW916: REAL := 40.0;  	(*температруа мойки 1 чистой водой*)
	TimeWashWater2_C2      		AT %MW918: DINT := 4;       	(*время мойки 2 чистой водой,мин*)
	TempWashWater2_C2      	AT %MW920: REAL := 40.0;  	(*температруа мойки 2 чистой водой*)
	TimeWashAlkaline_C2    		AT %MW922: DINT := 30;     	(*время мойки щелочью,мин*)
	TempWashAlkaline_C2    		AT %MW924: REAL := 75.0;  	(*температура мойки щелочью*)
	TimeAlkalineMix_C2     		AT %MW926: DINT := 60;     	(*время перемешивания при мойке щелочью,с*)
	TimeWashAcid_C2        		AT %MW928: DINT := 30;     	(*время мойки кислотой,мин*)
	TempWashAcid_C2        		AT %MW930: REAL := 65.0;  	(*температура мойки кислотой*)
	TimeAcidMix_C2         		AT %MW932: DINT := 60;     	(*время перемешивания при мойке кислотой,c*)
	TimeThermDesinf_C2     		AT %MW934: DINT := 10;      	(*время термической дезинфекции,мин*)
	TempThermDesinf_C2     		AT %MW936: REAL := 85.0;  	(*температура термической дезинфекции*)
	TempCoolThermDesinf_C2 	AT %MW938: REAL := 15.0;  	(*температура охлаждения терм дезинфекции*)
	TimeChemicDesinf_C2    		AT %MW940: DINT := 10;     	(*время химической дезинфекции,мин*)
	TimeSwillChemic_C2     		AT %MW942: DINT := 15;    	(*время ополаскивания чистой водой после хим дезинфекции*)
	TimeSwillWashWater1_C2    	AT %MW944: DINT := 5;  	(*время промывки водой со сбросом в Q4 после мойки 1 чистой водой,мин*)
	TimeSwillWashWater2_C2    	AT %MW946: DINT := 5;  	(*время промывки водой со сбросом в Q4 после мойки 2 чистой водой,мин*)

	(*рецепт*)
	RouteType_C2           		AT %MW970: DINT ;           	(*тип маршрута 1 - емкостной, 0 - замкнутый*)
	PumpCapacity_C2        		AT %MW972: DINT ;           	(*производительность подающего насоса *)
	TimeDelayRetPump_C2    	AT %MW974: DINT ;           	(*время задержки включения насоса возврата*)
	TimeDelayRetFlow_C2    		AT %MW976: DINT ;           	(*время появления протока на возврате*)
	TimeAlarmBackFlow_C2   		AT %MW978: DINT ;           	(*время аварии отсутствия обратного протока*)
	Numb_BackPump_C2       	AT %MW980: DINT ;           	(*номер насоса возврата*)
	VolumeDesinf_C2        		AT %MW982: DINT ;           	(*объем дезинфектанта*)
	Using_Q5_C2         			AT %MW984: DINT ;           	(*использование циркуляционного бака на мойках растворами и водой, 1 - использовать*)
	DeltaTempStartTime_C2  		AT %MW986: DINT ;           	(*перепад температуры TE1-TE2 для начала терм дезинфекции*)
	Route_C2               			AT %MW988: DINT ;           	(*номер выбранного маршрут контура*)

END_VAR

(* Global variable list: SolutionPrep *)
VAR_GLOBAL
	ModeQE_C1 	: INT; 	(*режим выбора пересчета концентрации, 0-щелочь, 1-кислота*)
	ModeQE_C2 	: INT; 	(*режим выбора пересчета концентрации, 0-щелочь, 1-кислота*)

END_VAR


VAR_GLOBAL RETAIN

	FlowPrep          		AT %MW1200: REAL := 20000;	(*производительность подающего насоса при подготовке*)
	TimeMixPrep       	AT %MW1202: DINT := 120;      	(*время перемешивания раствора в баке при подготовке,с*)
	EjectTime         		AT %MW1204: DINT := 20;      	(*время выталкивания щелочи (промывки) при подготовке*)

	MaxCondPrepAlk    	AT %MW1206: REAL := 1.95;    	(*максимальная проводимость раствора при подготовке щелочи*)
	MinCondPrepAlk    	AT %MW1208: REAL := 1.5;     	(*минимальная проводимость раствора при подготовке щелочи*)
	MaxTempPrepAlk    	AT %MW1210: REAL := 70.0;    	(*максимальная темп при подготовке щелочи*)
	MinTempPrepAlk    	AT %MW1212: REAL := 50.0;    	(*минимальная темп при подготовке щелочи*)
	LvlPrepAlk        		AT %MW1214: INT  := 65;      		(*заданный уровень в баке щелочи при подготовке*)

	MaxCondPrepAcid   	AT %MW1216: REAL := 1.3;     	(*максимальная проводимость раствора при подготовке кислоты*)
	MinCondPrepAcid   	AT %MW1218: REAL := 1.0;     	(*минимальная проводимость раствора при подготовке кислоты*)
	MaxTempPrepAcid  	AT %MW1220: REAL := 65.0;    	(*максимальная темп при подготовке кислоты*)
	MinTempPrepAcid  	AT %MW1222: REAL := 50.0;    	(*минимальная темп при подготовке кислоты*)
	LvlPrepAcid       		AT %MW1224: INT  := 65;      		(*заданный уровень в баке кислоты при подготовке*)

	Temp_etalonAlk    	AT %MW1226: REAL := 25.0;    	(*эталонная температура для щелочи*)
	Temp_etalonAcid   	AT %MW1228: REAL := 25.0;    	(*эталонная температура для кислоты*)
	Koef_tempAlk      	AT %MW1230: REAL := 0.0169;	(*температурный коэффициент щелочи (1/°С)*)
	Koef_tempAcid     	AT %MW1232: REAL := 0.0125;	(*температурный коэффициент кислоты (1/°С)*)
	QE_null_Alk       		AT %MW1234: REAL := 27.25;  	(*проводимость раствора щелочи при концентрации 0,5% и температуре T_etalonAlk (25гр)*)
	QE_null_Acid      	AT %MW1236: REAL := 29.3;    	(*проводимость раствора кислоты при концентрации 0,5% и температуре T_etalonAcid (25гр)*)
	Psi_Alk           		AT %MW1238: REAL := 52.5;    	(*коэффициент (изменение проводимости раствора щелочи при изменении его  концентрации на 1%)*)
	Psi_Acid          		AT %MW1240: REAL := 57.0;    	(*коэффициент (изменение проводимости раствора кислоты при изменении его  концентрации на 1%).*)
	CondAlk_Q4        	AT %MW1242: REAL := 1.1;     	(*концентрация для перехода с/на бак Q4*)
	CondAcid_Q4       	AT %MW1244: REAL := 0.75;    	(*концентрация для перехода с/на бак Q4*)




END_VAR

(* Global variable list: Timers *)
VAR_GLOBAL

	T_PowerLoss: TON; (* таймер перезапуска питания *)


END_VAR

(* Global variable list: Variable_Configuration *)
VAR_CONFIG RETAIN
	PLC_PRG.Kontur_1.Step                                                          	AT %MW1300 : INT;
	PLC_PRG.Kontur_1.Current_VolumeFC1                                   	AT %MW1302 : REAL;
	PLC_PRG.Kontur_1.Current_VolumeFC11                                 	AT %MW1304 : REAL;
	PLC_PRG.Kontur_1.Preparation.EjectionAlk                                                                	AT %MX1306.0 : BOOL;
	PLC_PRG.Kontur_1.Preparation.PastPrev                                 	AT %MW1308 : INT;
	PLC_PRG.Kontur_1.Preparation.Last_Time_min                        	AT %MW1310 : DINT;
	PLC_PRG.Kontur_1.Preparation.Last_Time_sec                        	AT %MW1312 : DINT;
	PLC_PRG.Kontur_1.Swill.PastPrev                                           	AT %MW1314 : INT;
	PLC_PRG.Kontur_1.Swill.StepBackPump                                  	AT %MW1316 : INT;
	PLC_PRG.Kontur_1.Swill.Step_Q4                                            	AT %MW1318 : INT;
	PLC_PRG.Kontur_1.Swill.Last_Time_min                                   	AT %MW1320 : DINT;
	PLC_PRG.Kontur_1.Swill.Last_Time_sec                                   	AT %MW1322 : DINT;
	PLC_PRG.Kontur_1.Swill.Return_Flow.Step                               	AT %MW1324 : INT;
	PLC_PRG.Kontur_1.Wash_Solution.PastPrev                            	AT %MW1326 : INT;
	PLC_PRG.Kontur_1.Wash_Solution.StepBackPump 				AT %MW1328 : INT;
	PLC_PRG.Kontur_1.Wash_Solution.Control_Q5.Step_Q5          	AT %MW1332 : INT;
	PLC_PRG.Kontur_1.Wash_Solution.Last_Time_min                   	AT %MW1334 : DINT;
	PLC_PRG.Kontur_1.Wash_Solution.Last_Time_sec                   	AT %MW1336 : DINT;
	PLC_PRG.Kontur_1.Wash_Solution.Preparation.EjectionAlk                               			AT %MX1306.1 : BOOL;
	PLC_PRG.Kontur_1.Wash_Solution.Preparation.PastPrev          	AT %MW1338 : INT;
	PLC_PRG.Kontur_1.Wash_Solution.Preparation.Last_Time_min	AT %MW1340 : DINT;
	PLC_PRG.Kontur_1.Wash_Solution.Preparation.Last_Time_sec	AT %MW1342 : DINT;
	PLC_PRG.Kontur_1.Wash_Solution.Return_Flow.Step               	AT %MW1344 : INT;
	PLC_PRG.Kontur_1.Wash_Water.Cool                                                                      		AT %MX1306.2 : BOOL;
	PLC_PRG.Kontur_1.Wash_Water.PastPrev                               	AT %MW1346 : INT;
	PLC_PRG.Kontur_1.Wash_Water.StepBackPump                      	AT %MW1348 : INT;
	PLC_PRG.Kontur_1.Wash_Water.Control_Q5.Step_Q5              	AT %MW1352 : INT;
	PLC_PRG.Kontur_1.Wash_Water.Last_Time_min                       	AT %MW1354 : DINT;
	PLC_PRG.Kontur_1.Wash_Water.Last_Time_sec                       	AT %MW1356 : DINT;
	PLC_PRG.Kontur_1.Wash_Water.Return_Flow.Step                   	AT %MW1358 : INT;
	PLC_PRG.Kontur_2.Step                                                          	AT %MW1360 : INT;
	PLC_PRG.Kontur_2.Current_VolumeFC1                                   	AT %MW1362 : REAL;
	PLC_PRG.Kontur_2.Current_VolumeFC11                                 	AT %MW1364 : REAL;
	PLC_PRG.Kontur_2.Preparation.EjectionAlk                                                             		AT %MX1306.3 : BOOL;
	PLC_PRG.Kontur_2.Preparation.PastPrev                                  	AT %MW1366 : INT;
	PLC_PRG.Kontur_2.Preparation.Last_Time_min                         	AT %MW1368 : DINT;
	PLC_PRG.Kontur_2.Preparation.Last_Time_sec                         	AT %MW1370 : DINT;
	PLC_PRG.Kontur_2.Swill.PastPrev                                            	AT %MW1372 : INT;
	PLC_PRG.Kontur_2.Swill.StepBackPump                                   	AT %MW1374 : INT;
	PLC_PRG.Kontur_2.Swill.Step_Q4                                             	AT %MW1376 : INT;
	PLC_PRG.Kontur_2.Swill.Last_Time_min                                    	AT %MW1378 : DINT;
	PLC_PRG.Kontur_2.Swill.Last_Time_sec                                    	AT %MW1380 : DINT;
	PLC_PRG.Kontur_2.Swill.Return_Flow.Step                                	AT %MW1382 : INT;
	PLC_PRG.Kontur_2.Wash_Solution.PastPrev                             	AT %MW1384 : INT;
	PLC_PRG.Kontur_2.Wash_Solution.StepBackPump                    	AT %MW1386 : INT;
	PLC_PRG.Kontur_2.Wash_Solution.Control_Q5.Step_Q5          	AT %MW1390 : INT;
	PLC_PRG.Kontur_2.Wash_Solution.Last_Time_min                   	AT %MW1392 : DINT;
	PLC_PRG.Kontur_2.Wash_Solution.Last_Time_sec                   	AT %MW1394 : DINT;
	PLC_PRG.Kontur_2.Wash_Solution.Preparation.EjectionAlk                                      		AT %MX1306.4 : BOOL;
	PLC_PRG.Kontur_2.Wash_Solution.Preparation.PastPrev          	AT %MW1396 : INT;
	PLC_PRG.Kontur_2.Wash_Solution.Preparation.Last_Time_min	AT %MW1398 : DINT;
	PLC_PRG.Kontur_2.Wash_Solution.Preparation.Last_Time_sec	AT %MW1400 : DINT;
	PLC_PRG.Kontur_2.Wash_Solution.Return_Flow.Step               	AT %MW1402 : INT;
	PLC_PRG.Kontur_2.Wash_Water.Cool                                                               			AT %MX1306.5 : BOOL;
	PLC_PRG.Kontur_2.Wash_Water.PastPrev                                  AT %MW1404 : INT;
	PLC_PRG.Kontur_2.Wash_Water.StepBackPump                      	AT %MW1406 : INT;
	PLC_PRG.Kontur_2.Wash_Water.Control_Q5.Step_Q5             	AT %MW1410 : INT;
	PLC_PRG.Kontur_2.Wash_Water.Last_Time_min                       	AT %MW1412 : DINT;
	PLC_PRG.Kontur_2.Wash_Water.Last_Time_sec                       	AT %MW1414 : DINT;
	PLC_PRG.Kontur_2.Wash_Water.Return_Flow.Step                   	AT %MW1416 : INT;


	PLC_PRG.Kontur_1.Chemical.PastPrev                                      	AT %MW1534 : INT;
	PLC_PRG.Kontur_1.Chemical.StepBackPump                             AT %MW1536 : INT;
	PLC_PRG.Kontur_1.Chemical.Last_Time_min 					AT %MW1538 : DINT;
	PLC_PRG.Kontur_1.Chemical.Last_Time_sec 					AT %MW1540 : DINT;
	PLC_PRG.Kontur_1.Chemical.Return_Flow.Step 				AT %MW1542 : INT;
	PLC_PRG.Kontur_1.Chemical.Control_Q5.Step_Q5 				AT %MW1544 : INT;
	PLC_PRG.Kontur_2.Chemical.PastPrev 						AT %MW1546 : INT;
	PLC_PRG.Kontur_2.Chemical.StepBackPump 					AT %MW1548 : INT;
	PLC_PRG.Kontur_2.Chemical.Last_Time_min 					AT %MW1550 : DINT;
	PLC_PRG.Kontur_2.Chemical.Last_Time_sec 					AT %MW1552 : DINT;
	PLC_PRG.Kontur_2.Chemical.Return_Flow.Step 				AT %MW1554 : INT;
	PLC_PRG.Kontur_2.Chemical.Control_Q5.Step_Q5 				AT %MW1556 : INT;

END_VAR

(* Global variable list: Visualisations *)
VAR_GLOBAL

(*-----------------------Общие------------------------------*)
	Vis_ConcAlk_alarm		AT %QX468.0 	: BOOL;		(*визуализация датчика аварийного нижнего уровня в баке концентрата щелочи Q7*)
	Vis_ConcAlk_min		AT %QX468.1 	: BOOL;		(*визуализация датчика нижнего уровня в баке концентрата щелочи Q7*)
	Vis_ConcAcid_alarm		AT %QX468.2 	: BOOL;		(*визуализация датчика аварийного нижнего уровня в баке концентрата кислоты Q8*)
	Vis_ConcAcid_min		AT %QX468.3 	: BOOL;		(*визуализация датчика нижнего уровня в баке концентрата кислоты Q8*)
	Vis_PS1					AT %QX468.4 	: BOOL;		(*визуализация датчика давления сжатого воздуха*)
(*-----------------------контур 1---------------------------*)
	Vis_tim_Process_C1    	AT %QX470.0 	: BOOL;		(*визуализация полей времени*)
	Change_Mode_C1        	AT %QX470.1 	: BOOL; 	(*сигнал в ОР что режим не выбран*)
	Vis_ManMode_C1      	AT %QX470.2 	: BOOL; 	(*сигнал в ОР что выбран ручной режим*)
	Vis_Pause_C1             	AT %QX470.3	: BOOL; 	(*визуализации кнопки пауза мойки*)
	Vis_PrepAlk_C1            	AT %QX470.4	: BOOL;  	(*визуализации кнопки подготовки р-ра*)
	Vis_PrepAcid_C1       	AT %QX470.5	: BOOL;  	(*визуализации кнопки подготовки р-ра*)
	Vis_RouteReady_K1    	AT %QX470.6	: BOOL; 	(*визуализации готовности выбранного маршрута по контуру 1*)
	Vis_FS_K1    			AT %QX470.7	: BOOL; 	(*визуализация датчика протока на возврате по контуру 1*)
	Vis_LSL_K1    			AT %QX470.8	: BOOL; 	(*визуализация датчика нижнего уровня в цирк баке  контура 1*)
	Vis_LSM_K1    			AT %QX470.9	: BOOL; 	(*визуализация датчика среднего уровня в цирк баке  контура 1*)
	Vis_LSH_K1    			AT %QX470.10	: BOOL; 	(*визуализация датчика верхнего уровня в цирк баке  контура 1*)

	Vis_Pipe_C1_1			AT%QW471	: WORD;		(*визуализация труб*)
	Vis_Pipe_C1_2			AT%QW472	: WORD;		(*визуализация труб*)
	w_Step_C1                     	AT%QW473 	: WORD;		(*шаги работы контура - побитно*)
	Step_C1               		AT%QW474	: INT;  			(*шаги работы контура*)
	VisuMode_C1          		AT%QW475	: INT;			(*текущая стадия работы*)
	Last_Time_min_C1      	AT%QW476	: DINT;  			(*расчет оставшихся минут процесса*)
	Last_Time_sec_C1      	AT%QW478	: DINT;  			(*расчет оставшихся секунд процесса*)


(*---------------------контур 2--------------------------------*)
	Vis_tim_Process_C2    	AT %QX480.0 	: BOOL; 	(*визуализация полей времени*)
	Change_Mode_C2        	AT %QX480.1 	: BOOL; 	(*сигнал в ОР что режим не выбран*)
	Vis_ManMode_C2         	AT %QX480.2 	: BOOL; 	(*сигнал в ОР что выбран ручной режим*)
	Vis_Pause_C2              	AT %QX480.3	: BOOL; 	(*визуализации кнопки пауза мойки*)
	Vis_PrepAlk_C2            	AT %QX480.4	: BOOL;  	(*визуализации кнопки подготовки р-ра*)
	Vis_PrepAcid_C2         	AT %QX480.5	: BOOL;  	(*визуализации кнопки подготовки р-ра*)
	Vis_RouteReady_K2    	AT %QX480.6	: BOOL; 	(*визуализации готовности выбранного маршрута по контуру 2*)
	Vis_FS_K2    			AT %QX480.7	: BOOL; 	(*визуализация датчика протока на возврате по контуру 2*)
	Vis_LSL_K2    			AT %QX480.8	: BOOL; 	(*визуализация датчика нижнего уровня в цирк баке  контура 2*)
	Vis_LSM_K2    			AT %QX480.9	: BOOL; 	(*визуализация датчика среднего уровня в цирк баке  контура 2*)
	Vis_LSH_K2    			AT %QX480.10	: BOOL; 	(*визуализация датчика верхнего уровня в цирк баке  контура 2*)

	Vis_Pipe_C2_1			AT%QW481	: WORD;	(*визуализация труб*)
	Vis_Pipe_C2_2			AT%QW482	: WORD;	(*визуализация труб*)
	w_Step_C2                     	AT%QW483 	: WORD;  	(*шаги работы контура - побитно*)
	Step_C2              		AT%QW484	:  INT;  		(*шаги работы контура*)
	VisuMode_C2           		AT%QW485	:  INT;		(*текущая стадия работы*)
	Last_Time_min_C2      	AT%QW486	: DINT;  		(*расчет оставшихся минут процесса*)
	Last_Time_sec_C2      	AT%QW488	: DINT;  		(*расчет оставшихся секунд процесса*)

(*---------------------контур 3--------------------------------*)
(*%QX490 - %QX498*)

END_VAR

(* POU PLC_PRG, ST *)
PROGRAM PLC_PRG
VAR
   first_scan :BOOL:=FALSE;   (*первый скан-0, потом постоянно-1*)
   fb_SystemTime :TimerIncr ; (*определение системного времени*)

   Kontur_1:Circuit;
   Kontur_2:Circuit;



END_VAR
(*определение запуска плк*)
 IF NOT first_scan THEN
    Power_loss := TRUE;
    T_PowerLoss.in := TRUE;
 END_IF;
 IF T_PowerLoss.q THEN
     Power_loss := FALSE;
     T_PowerLoss.in :=FALSE;
 END_IF;
T_PowerLoss(PT:=T#15s);


fb_SystemTime(q_scan_time=>scan_time); (*системное время в мс*)
Inputs();
AlarmReaction();

(*обнуление общих механизмов в начале скана*)
	q_VA1   := FALSE;
	q_VE7  := FALSE;
	q_P8  := FALSE;
	q_P9  := FALSE;

     q_Green :=FALSE;
     q_Yellow :=FALSE;
     q_Red:=FALSE;
     q_Sirena :=FALSE;

  H1_q:=FALSE;
  H2_q:=FALSE;
  H3_q:=FALSE;
  H4_q:=FALSE;
  H5_q:=FALSE;
  H6_q:=FALSE;
  H7_q:=FALSE;
  H8_q:=FALSE;
  H9_q:=FALSE;


(*---------------Контур 1--------------------------*)

Kontur_1.i_DiagSwillBackWater:=Alarm_PS OR Alarm_PE1 OR Alarm_Stop OR Power_loss OR Alarm_FE11 OR AlarmBackFlow_C1
                                        OR Alarm_MinLev_Q1 OR Alarm_VA541 OR Alarm_VA401 OR Alarm_VA41 OR Alarm_VA11
                                        OR Alarm_VA531 OR Alarm_P1;
Kontur_1.i_DiagSwillFreshWater:=Alarm_PS OR Alarm_PE1 OR Alarm_Stop OR Power_loss OR Alarm_FE11 OR AlarmBackFlow_C1
                                         OR Alarm_MinLev_Q1 OR Alarm_VA541 OR Alarm_VA401  OR Alarm_VA11
                                         OR Alarm_VA531 OR Alarm_P1;
Kontur_1.i_DiagWashAlkaline:=Alarm_PS OR Alarm_PE1 OR Alarm_Stop OR Power_loss OR Alarm_FE11 OR AlarmBackFlow_C1
                                      OR Alarm_MinLev_Q1 OR Alarm_MinLev_Q2 OR Alarm_VA541 OR Alarm_VA401 OR Alarm_VA201
                                      OR Alarm_VA11 OR Alarm_VA21 OR Alarm_VA5 OR Alarm_VA501 OR Alarm_VA51 OR Alarm_VA521
                                      OR Alarm_VA531 OR Alarm_P1;
Kontur_1.i_DiagWashAcid:=Alarm_PS OR Alarm_PE1 OR Alarm_Stop OR Power_loss OR Alarm_FE11 OR AlarmBackFlow_C1
                                  OR Alarm_MinLev_Q1 OR Alarm_MinLev_Q3 OR Alarm_VA541 OR Alarm_VA401 OR Alarm_VA301
                                  OR Alarm_VA11 OR Alarm_VA31 OR Alarm_VA5 OR Alarm_VA501 OR Alarm_VA51 OR Alarm_VA521
                                  OR Alarm_VA531 OR Alarm_P1;
Kontur_1.i_DiagWashWater:=Alarm_PS OR Alarm_PE1 OR Alarm_Stop OR Power_loss OR Alarm_FE11 OR AlarmBackFlow_C1
                                   OR Alarm_MinLev_Q1 OR Alarm_VA541 OR Alarm_VA401 OR Alarm_VA11 OR Alarm_VA5
                                   OR Alarm_VA501 OR Alarm_VA51 OR Alarm_VA531 OR Alarm_P1;
Kontur_1.i_DiagThermDesinfection:=Alarm_PS OR Alarm_PE1 OR Alarm_Stop OR Power_loss OR Alarm_FE11 OR AlarmBackFlow_C1
                                           OR Alarm_MinLev_Q1 OR Alarm_VA541 OR Alarm_VA401 OR Alarm_VA11 OR Alarm_VA5
                                           OR Alarm_VA501 OR Alarm_VA51 OR Alarm_VA531 OR Alarm_P1;
Kontur_1.i_DiagChemicDesinfection:=Alarm_PS OR Alarm_PE1 OR Alarm_Stop OR Power_loss OR Alarm_FE11 OR AlarmBackFlow_C1
                                            OR Alarm_MinLev_Q1 OR Alarm_VA541 OR Alarm_VA401 OR Alarm_VA11 OR Alarm_VA5
                                            OR Alarm_VA501 OR Alarm_VA51 OR Alarm_VA531 OR Alarm_P1 ;
Kontur_1.i_DiagPrepareAlkaline:=Alarm_PS OR Alarm_PE1 OR Alarm_Stop OR Power_loss OR Alarm_FE11
                                         OR Alarm_MinLev_Q1 OR Alarm_VA541 OR Alarm_VA401 OR Alarm_VA201
                                         OR Alarm_VA11 OR Alarm_VA21  OR Alarm_VA521
                                         OR Alarm_VA531 OR Alarm_P1 ;
Kontur_1.i_DiagPrepareAcid:=Alarm_PS OR Alarm_PE1 OR Alarm_Stop OR Power_loss OR Alarm_FE11
                                         OR Alarm_MinLev_Q1 OR Alarm_VA541 OR Alarm_VA401 OR Alarm_VA301
                                         OR Alarm_VA11 OR Alarm_VA31  OR Alarm_VA521
                                         OR Alarm_VA531 OR Alarm_P1 ;
Kontur_1.i_DiagHandMode:= Alarm_PS OR Alarm_Stop OR Power_loss;
Kontur_1.i_DiagDiagnostic:=Alarm_PS OR Alarm_Stop OR Power_loss;

Kontur_1(
	w_ManDevice:=w_ManDevice_C1 ,
	Man_VE7:=Man_VE7,
	Man_P8:=Man_P8,
	Man_P9:=Man_P9,
	Man_P10:=Man_P10,
	ManSP_P1:=ManSP_P1,
	ManSP_VR1:=ManSP_VR1,

	i_Block_Q4_out:=	FALSE ,      (*используем для режима нейтрализации перед сбросом моющих*)
	i_Block_Q4_in_level:= FALSE , (*используем для режима нейтрализации перед сбросом моющих*)
      	i_Block_Q4_in_ph:= FALSE , 	(*используем для режима нейтрализации перед сбросом моющих*)
	i_Ready_Route:= TRUE  ,		(*используем для системы с контролем готовности выбранного маршрута*)

	i_Block_SolPrep_Alk:=(Kontur_2.Step=6) ,
	i_Block_SolPrep_Acid:=(Kontur_2.Step=10)  ,
	i_Block_Wash_Alk:=Kontur_2.q_Block_Solution_Alk  ,
	i_Block_Wash_Acid:=Kontur_2.q_Block_Solution_Acid  ,
	i_Alarm_LSmin_Alk:=Alarm_LS71 ,
	i_Alarm_LSmin_Acid:=Alarm_LS81 ,
	i_Alarm_LSmin_Dez:= TRUE ,	(*используем при работе с хим дезинфекцией*)
	i_Alarm_PE:=Alarm_PE1 ,

	i_Pause:=Pause_C1 ,
	i_Stop:=Stop_C1 ,
	i_Start_AutoWashing:=Start_AutoWashing_C1 AND (Route_C1 <> 0),  (*запуск мойки в автомате при выбранном маршруте*)
	i_Start_HandMode:=Start_HandMode_C1  ,
	i_Start_PrepareAlkaline:=Start_PrepareAlkaline_C1 ,
	i_Start_PrepareAcid:=Start_PrepareAcid_C1 ,
	i_Start_Diagnostic:=Start_Diagnostic_C1 ,
	i_ch_SwillBackWater:=ch_SwillBackWater_C1 ,
	i_ch_SwillFreshWater:=ch_SwillFreshWater_C1 ,
	i_ch_WashAlkaline:=ch_WashAlkaline_C1 ,
	i_ch_WashWater1:=ch_WashWater1_C1 ,
	i_ch_WashAcid:=ch_WashAcid_C1 ,
	i_ch_WashWater2:=ch_WashWater2_C1 ,
	i_ch_ThermDesinfection:=ch_ThermDesinfection_C1 ,
	i_ch_ChemicDesinfection:=ch_ChemicDesinfection_C1 ,
	i_FS1:= ,					(*используем при работе с хим дезинфекцией*)
	i_FC11:=FC1_i ,
	i_FS:=FS21_i ,
	i_LSL:=LSL5_i ,
	i_LSM:=LSM5_i ,
	i_LSH:=LSH5_i ,
	i_TE1:=i_TE11 ,
	i_TE2:=i_TE21 ,
	i_TE_Q2:=i_TE2 ,
	i_LE_Q2:=i_LE2 ,
	i_TE_Q3:=i_TE3 ,
	i_LE_Q3:=i_LE3 ,
	i_QE:=QE1 ,
	i_QE_priv:=QE1_priv ,

	i_TimeDelay:=TimeDelay_C1 ,
	i_Time_LSH_on:=Time_LSH_on ,
	i_Time_LSM_on:=Time_LSM_on ,
	i_Time_LSM_off:=Time_LSM_off ,
	i_Time_LSL_off:=Time_LSL_off ,
	i_K_imp:=K_imp_C1 ,
	i_K_imp_dez:=K_imp_dez_C1 ,		(*используем при работе с хим дезинфекцией*)

	i_AlkMixing:=AlkMixing_C1  ,
	i_AcidMixing:=AcidMixing_C1 ,

	i_TimeSwillBackWater:=TimeSwillBackWater_C1 ,
	i_TimeSwillFreshWater:=TimeSwillFreshWater_C1 ,
	i_TimeWashWater1:=TimeWashWater1_C1 ,
      	i_TimeSwillWashWater1:=TimeSwillWashWater1_C1 ,
	i_TempWashWater1:=TempWashWater1_C1 ,
	i_TimeWashWater2:=TimeWashWater2_C1 ,
       i_TimeSwillWashWater2:=TimeSwillWashWater2_C1 ,
	i_TempWashWater2:=TempWashWater2_C1 ,
	i_TimeWashAlkaline:=TimeWashAlkaline_C1 ,
	i_TempWashAlkaline:=TempWashAlkaline_C1 ,
	i_TimeWashAcid:=TimeWashAcid_C1 ,
	i_TempWashAcid:=TempWashAcid_C1  ,
	i_TimeThermDesinf:=TimeThermDesinf_C1 ,
	i_TempThermDesinf:=TempThermDesinf_C1 ,
	i_TempCoolThermDesinf:=TempCoolThermDesinf_C1 ,
	i_TimeChemicDesinf:=TimeChemicDesinf_C1 ,
	i_TimeSwillChemic:=TimeSwillChemic_C1 ,

	i_RouteType:=RouteType_C1 ,
	i_PumpCapacity:=PumpCapacity_C1 ,
	i_TimeDelayRetPump:=TimeDelayRetPump_C1 ,
	i_TimeDelayRetFlow:=TimeDelayRetFlow_C1 ,
	i_TimeAlarmBackFlow:=TimeAlarmBackFlow_C1 ,
	i_Numb_BackPump:=Numb_BackPump_C1 ,
	i_VolumeDesinf:=VolumeDesinf_C1 ,			(*используем при работе с хим дезинфекцией*)
       i_Using_Q5 := Using_Q5_C1 ,
	i_DeltaTempStartTime:=DeltaTempStartTime_C1 ,

	w_qDevice=> w_qDevice_C1 ,

	q_Vis_tim_Process=>Vis_tim_Process_C1 ,
	q_Change_Mode=>Change_Mode_C1 ,
	q_Run_Process=>  ,					(*используем для системы с контролем готовности выбранного маршрута*)

	q_SP_P1=>SP_P1 ,
	q_SP_VR1=>SP_VR1 ,
	q_VisuMode=>VisuMode_C1 ,
	q_ModeQE=>ModeQE_C1 ,
	q_Last_Time_min=>Last_Time_min_C1 ,
	q_Last_Time_sec=>Last_Time_sec_C1 );

    Step_C1 := Kontur_1.Step;
    Current_VolumeFC1 := Kontur_1.Current_VolumeFC1;
    Current_VolumeFC11 := Kontur_1.Current_VolumeFC11;
    Vis_ManMode_C1 := (Kontur_1.Step=18); (*визуализация кнопок ручного режима*)
    Vis_Pause_C1 := Kontur_1.Step<>0 AND Kontur_1.Step<>18 AND Kontur_1.Step<>21; (*визуализации кнопки пауза мойки*)
    	IF Kontur_1.Step=0 THEN
      		Pause_C1 := FALSE;
    	END_IF;
    (*виз кнопока запуска подготовки растворов*)
	Vis_PrepAlk_C1  := Change_Mode_C1 AND NOT ((Kontur_2.Step=6)    OR (Kontur_2.Step=19));
	Vis_PrepAcid_C1:= Change_Mode_C1 AND NOT ((Kontur_2.Step=10)  OR (Kontur_2.Step=20));

	IF Kontur_1.q_AlarmBackFlow THEN (*Нет протока на возврате*)
       	AlarmBackFlow_C1:=TRUE;
  	END_IF;
	IF Kontur_1.q_Alarm_Empty_Q5 THEN (*авария опустошения цирк бака при работе на замкн маршруте*)
   		Alarm_Empty_Q5:=TRUE;
    	END_IF;
    	IF Kontur_1.T_Control_TE.Q THEN (*Долгий нагрев*)
  		HeatingAlarm_C1 := TRUE;
    	END_IF;
    	IF Kontur_1.T_Control_QE.Q THEN (*Долгий набор концентрации*)
      		CondAlarm_C1 := TRUE;
    	END_IF;

	(*обнуление номера маршрута при окончании мойки в автомате*)
	IF Kontur_1.q_End_AutoMode THEN
		Route_C1 := 0;
	END_IF;

(*выбор насоса возврата*)
CASE Numb_BackPump_C1 OF
0:;
1:
  H1_q:=w_qDevice_C1.BackPump;
2:
  H2_q:=w_qDevice_C1.BackPump;
3:
  H3_q:=w_qDevice_C1.BackPump;
4:
  H4_q:=w_qDevice_C1.BackPump;
5:
  H5_q := w_qDevice_C1.BackPump;
6:
  H6_q:=w_qDevice_C1.BackPump;
7:
  H7_q:=w_qDevice_C1.BackPump;
8:
  H8_q:=w_qDevice_C1.BackPump;
9:
  H9_q:=w_qDevice_C1.BackPump;
ELSE
	Numb_BackPump_C1 := 5; (*номер насоса возврата по умолчанию для контура*)
END_CASE;

(*обнуление кнопок ручного режима*)
IF Kontur_1.Step=0 THEN
	w_ManDevice_C1 := 0;
	ManSP_P1 := 0.0;
	ManSP_VR1 := 0.0;
END_IF;

(*-------------------------------------------------*)



(*---------------Контур 2--------------------------*)

Kontur_2.i_DiagSwillBackWater:=Alarm_PS OR Alarm_PE2 OR Alarm_Stop OR Power_loss OR Alarm_FE12 OR AlarmBackFlow_C2
                                        OR Alarm_MinLev_Q1 OR Alarm_VA642 OR Alarm_VA402 OR Alarm_VA42 OR Alarm_VA12
                                        OR Alarm_VA632 OR Alarm_P2;
Kontur_2.i_DiagSwillFreshWater:=Alarm_PS OR Alarm_PE2 OR Alarm_Stop OR Power_loss OR Alarm_FE12 OR AlarmBackFlow_C2
                                         OR Alarm_MinLev_Q1 OR Alarm_VA642 OR Alarm_VA402  OR Alarm_VA12
                                         OR Alarm_VA632 OR Alarm_P2;
Kontur_2.i_DiagWashAlkaline:=Alarm_PS OR Alarm_PE2 OR Alarm_Stop OR Power_loss OR Alarm_FE12 OR AlarmBackFlow_C2
                                      OR Alarm_MinLev_Q1 OR Alarm_MinLev_Q2 OR Alarm_VA642 OR Alarm_VA402 OR Alarm_VA202
                                      OR Alarm_VA12 OR Alarm_VA22 OR Alarm_VA6 OR Alarm_VA602 OR Alarm_VA62 OR Alarm_VA622
                                      OR Alarm_VA632 OR Alarm_P2;
Kontur_2.i_DiagWashAcid:=Alarm_PS OR Alarm_PE2 OR Alarm_Stop OR Power_loss OR Alarm_FE12 OR AlarmBackFlow_C2
                                  OR Alarm_MinLev_Q1 OR Alarm_MinLev_Q3 OR Alarm_VA642 OR Alarm_VA402 OR Alarm_VA302
                                  OR Alarm_VA12 OR Alarm_VA32 OR Alarm_VA6 OR Alarm_VA602 OR Alarm_VA62 OR Alarm_VA622
                                  OR Alarm_VA632 OR Alarm_P2;
Kontur_2.i_DiagWashWater:=Alarm_PS OR Alarm_PE2 OR Alarm_Stop OR Power_loss OR Alarm_FE12 OR AlarmBackFlow_C2
                                   OR Alarm_MinLev_Q1 OR Alarm_VA642 OR Alarm_VA402 OR Alarm_VA12 OR Alarm_VA6
                                   OR Alarm_VA602 OR Alarm_VA62 OR Alarm_VA632 OR Alarm_P2;
Kontur_2.i_DiagThermDesinfection:=Alarm_PS OR Alarm_PE2 OR Alarm_Stop OR Power_loss OR Alarm_FE12 OR AlarmBackFlow_C2
                                           OR Alarm_MinLev_Q1 OR Alarm_VA642 OR Alarm_VA402 OR Alarm_VA12 OR Alarm_VA6
                                           OR Alarm_VA602 OR Alarm_VA62 OR Alarm_VA632 OR Alarm_P2;
Kontur_2.i_DiagChemicDesinfection:=Alarm_PS OR Alarm_PE2 OR Alarm_Stop OR Power_loss OR Alarm_FE12 OR AlarmBackFlow_C2
                                            OR Alarm_MinLev_Q1 OR Alarm_VA642 OR Alarm_VA402 OR Alarm_VA12 OR Alarm_VA6
                                            OR Alarm_VA602 OR Alarm_VA62 OR Alarm_VA632 OR Alarm_P2 ;
Kontur_2.i_DiagPrepareAlkaline:=Alarm_PS OR Alarm_PE2 OR Alarm_Stop OR Power_loss OR Alarm_FE12
                                         OR Alarm_MinLev_Q1 OR Alarm_VA642 OR Alarm_VA402 OR Alarm_VA202
                                         OR Alarm_VA12 OR Alarm_VA22  OR Alarm_VA622
                                         OR Alarm_VA632 OR Alarm_P2 ;
Kontur_2.i_DiagPrepareAcid:=Alarm_PS OR Alarm_PE2 OR Alarm_Stop OR Power_loss OR Alarm_FE12
                                         OR Alarm_MinLev_Q1 OR Alarm_VA642 OR Alarm_VA402 OR Alarm_VA302
                                         OR Alarm_VA12 OR Alarm_VA32  OR Alarm_VA622
                                         OR Alarm_VA632 OR Alarm_P2 ;
Kontur_2.i_DiagHandMode:= Alarm_PS OR Alarm_Stop OR Power_loss;
Kontur_2.i_DiagDiagnostic:=Alarm_PS OR Alarm_Stop OR Power_loss;

Kontur_2(
	w_ManDevice:=w_ManDevice_C2 ,
	Man_VE7:=Man_VE7,
	Man_P8:=Man_P8,
	Man_P9:=Man_P9,
	Man_P10:=Man_P10,
	ManSP_P1:=ManSP_P2,
	ManSP_VR1:=ManSP_VR2,

	i_Block_Q4_out:=	FALSE ,      (*используем для режима нейтрализации перед сбросом моющих*)
	i_Block_Q4_in_level:= FALSE , (*используем для режима нейтрализации перед сбросом моющих*)
      	i_Block_Q4_in_ph:= FALSE , 	(*используем для режима нейтрализации перед сбросом моющих*)
	i_Ready_Route:= TRUE  ,		(*используем для системы с контролем готовности выбранного маршрута*)

	i_Block_SolPrep_Alk:=(Kontur_1.Step=6) ,
	i_Block_SolPrep_Acid:=(Kontur_1.Step=10)  ,
	i_Block_Wash_Alk:=Kontur_1.q_Block_Solution_Alk  ,
	i_Block_Wash_Acid:=Kontur_1.q_Block_Solution_Acid  ,
	i_Alarm_LSmin_Alk:=Alarm_LS71 ,
	i_Alarm_LSmin_Acid:=Alarm_LS81 ,
	i_Alarm_LSmin_Dez:= TRUE ,	(*используем при работе с хим дезинфекцией*)
	i_Alarm_PE:=Alarm_PE2 ,

	i_Pause:=Pause_C2 ,
	i_Stop:=Stop_C2 ,
	i_Start_AutoWashing:=Start_AutoWashing_C2 AND (Route_C2 <> 0),  (*запуск мойки в автомате при выбранном маршруте*)
	i_Start_HandMode:=Start_HandMode_C2  ,
	i_Start_PrepareAlkaline:=Start_PrepareAlkaline_C2 ,
	i_Start_PrepareAcid:=Start_PrepareAcid_C2 ,
	i_Start_Diagnostic:=Start_Diagnostic_C2 ,
	i_ch_SwillBackWater:=ch_SwillBackWater_C2 ,
	i_ch_SwillFreshWater:=ch_SwillFreshWater_C2 ,
	i_ch_WashAlkaline:=ch_WashAlkaline_C2 ,
	i_ch_WashWater1:=ch_WashWater1_C2 ,
	i_ch_WashAcid:=ch_WashAcid_C2 ,
	i_ch_WashWater2:=ch_WashWater2_C2 ,
	i_ch_ThermDesinfection:=ch_ThermDesinfection_C2 ,
	i_ch_ChemicDesinfection:=ch_ChemicDesinfection_C2 ,

	i_FS1:= ,							(*используем при работе с хим дезинфекцией*)
	i_FC11:=FC2_i ,
	i_FS:=FS22_i ,
	i_LSL:=LSL6_i ,
	i_LSM:=LSM6_i ,
	i_LSH:=LSH6_i ,

	i_TE1:=i_TE12 ,
	i_TE2:=i_TE22 ,
	i_TE_Q2:=i_TE2 ,
	i_LE_Q2:=i_LE2 ,
	i_TE_Q3:=i_TE3 ,
	i_LE_Q3:=i_LE3 ,
	i_QE:=QE2 ,
	i_QE_priv:=QE2_priv ,

	i_TimeDelay:=TimeDelay_C2 ,
	i_Time_LSH_on:=Time_LSH_on ,
	i_Time_LSM_on:=Time_LSM_on ,
	i_Time_LSM_off:=Time_LSM_off ,
	i_Time_LSL_off:=Time_LSL_off ,
	i_K_imp:=K_imp_C2 ,
	i_K_imp_dez:=K_imp_dez_C2 ,	(*используем при работе с хим дезинфекцией*)

	i_AlkMixing:=AlkMixing_C2  ,
	i_AcidMixing:=AcidMixing_C2 ,

	i_TimeSwillBackWater:=TimeSwillBackWater_C2 ,
	i_TimeSwillFreshWater:=TimeSwillFreshWater_C2 ,
	i_TimeWashWater1:=TimeWashWater1_C2 ,
      i_TimeSwillWashWater1:=TimeSwillWashWater1_C2 ,
	i_TempWashWater1:=TempWashWater1_C2 ,
	i_TimeWashWater2:=TimeWashWater2_C2 ,
      i_TimeSwillWashWater2:=TimeSwillWashWater2_C2 ,
	i_TempWashWater2:=TempWashWater2_C2 ,
	i_TimeWashAlkaline:=TimeWashAlkaline_C2 ,
	i_TempWashAlkaline:=TempWashAlkaline_C2 ,
	i_TimeWashAcid:=TimeWashAcid_C2 ,
	i_TempWashAcid:=TempWashAcid_C2  ,
	i_TimeThermDesinf:=TimeThermDesinf_C2 ,
	i_TempThermDesinf:=TempThermDesinf_C2 ,
	i_TempCoolThermDesinf:=TempCoolThermDesinf_C2 ,
	i_TimeChemicDesinf:=TimeChemicDesinf_C2 ,
	i_TimeSwillChemic:=TimeSwillChemic_C2 ,

	i_RouteType:=RouteType_C2 ,
	i_PumpCapacity:=PumpCapacity_C2 ,
	i_TimeDelayRetPump:=TimeDelayRetPump_C2 ,
	i_TimeDelayRetFlow:=TimeDelayRetFlow_C2 ,
	i_TimeAlarmBackFlow:=TimeAlarmBackFlow_C2 ,
	i_Numb_BackPump:=Numb_BackPump_C2 ,
	i_VolumeDesinf:=VolumeDesinf_C2 ,
       i_Using_Q5 := Using_Q5_C2 ,
	i_DeltaTempStartTime:=DeltaTempStartTime_C2 ,

	w_qDevice=> w_qDevice_C2 ,

	q_Vis_tim_Process=>Vis_tim_Process_C2 ,
	q_Change_Mode=>Change_Mode_C2 ,

	q_Run_Process=>  ,					(*используем для системы с контролем готовности выбранного маршрута*)

	q_SP_P1=>SP_P2 ,
	q_SP_VR1=>SP_VR2 ,
	q_VisuMode=>VisuMode_C2 ,
	q_ModeQE=>ModeQE_C2 ,
	q_Last_Time_min=>Last_Time_min_C2 ,
	q_Last_Time_sec=>Last_Time_sec_C2 );

    Step_C2 := Kontur_2.Step;
    Current_VolumeFC2 := Kontur_2.Current_VolumeFC1;
    Current_VolumeFC12 := Kontur_2.Current_VolumeFC11;
    Vis_ManMode_C2 := (Kontur_2.Step=18); (*визуализация кнопок ручного режима*)
    Vis_Pause_C2 := Kontur_2.Step<>0 AND Kontur_2.Step<>18 AND Kontur_2.Step<>21; (*визуализации кнопки пауза мойки*)
    IF Kontur_2.Step = 0 THEN
     	 Pause_C2 := FALSE;
    END_IF;
    (*виз кнопок запуска подготовки растворов*)
	Vis_PrepAlk_C2   := Change_Mode_C2 AND NOT ((Kontur_1.Step=6)  OR (Kontur_1.Step=19));
	Vis_PrepAcid_C2 := Change_Mode_C2 AND NOT ((Kontur_1.Step=10) OR (Kontur_1.Step=20) );

	IF Kontur_2.q_AlarmBackFlow THEN (*Нет протока на возврате*)
       	AlarmBackFlow_C2 := TRUE;
    	END_IF;
	IF Kontur_2.q_Alarm_Empty_Q5 THEN (*авария опустошения цирк бака при работе на замкн маршруте*)
       	Alarm_Empty_Q6 := TRUE;
    	END_IF;
    	IF Kontur_2.T_Control_TE.Q THEN (*Долгий нагрев*)
       	HeatingAlarm_C2 := TRUE;
    	END_IF;
   	 IF Kontur_2.T_Control_QE.Q THEN (*Долгий набор концентрации*)
       	CondAlarm_C2:=TRUE;
    	END_IF;

	(*обнуление номера маршрута при окончании мойки в автомате*)
	IF Kontur_2.q_End_AutoMode THEN
		Route_C2 := 0;
	END_IF;

(*выбор насоса возврата*)
CASE Numb_BackPump_C2 OF
0:;
1:
  H1_q:=w_qDevice_C2.BackPump;
2:
  H2_q:=w_qDevice_C2.BackPump;
3:
  H3_q:=w_qDevice_C2.BackPump;
4:
  H4_q:=w_qDevice_C2.BackPump;
5:
  H5_q:=w_qDevice_C2.BackPump;
6:
  H6_q:=w_qDevice_C2.BackPump;
7:
  H7_q:=w_qDevice_C2.BackPump;
8:
  H8_q:=w_qDevice_C2.BackPump;
9:
  H9_q:=w_qDevice_C2.BackPump;
ELSE
	Numb_BackPump_C2 := 1; (*номер насоса возврата по умолчанию для контура*)
END_CASE;

(*обнуление кнопок ручного режима*)
IF Kontur_2.Step=0 THEN
	w_ManDevice_C2 := 0;
	ManSP_P2:=0.0;
	ManSP_VR2:=0.0;
END_IF;

(*-------------------------------------------------*)


(*-------------------------------------------------*)
(*обнуление кнопок ручного режима для общих механизмов*)
IF Kontur_1.Step<>18 AND Kontur_2.Step<>18   THEN
	Man_VE7 := FALSE;
	Man_P8 := FALSE;
	Man_P9 := FALSE;
END_IF;

(*---------------общие механизмы----------------*)
	q_VE7 :=Kontur_1.q_VE7 OR Kontur_2.q_VE7 ;
	q_P8   :=Kontur_1.q_P8  OR Kontur_2.q_P8  ;
	q_P9   :=Kontur_1.q_P9  OR Kontur_2.q_P9  ;
	q_P10   :=Kontur_1.q_P10  OR Kontur_2.q_P10  ;

	q_Red :=    Kontur_1.q_Red       OR Kontur_2.q_Red  ;
	q_Yellow := Kontur_1.q_Yellow  OR Kontur_2.q_Yellow  ;
	q_Green  :=Kontur_1.q_Green   OR Kontur_2.q_Green   ;
	q_Sirena :=Kontur_1.q_Sirena  OR Kontur_2.q_Sirena  ;
(*-------------------------------------------------*)





DeviceControl();
Visualisation();



first_scan:=TRUE; (*флаг определения первого скана, взводится в конце первого скана*)
END_PROGRAM

(* POU Circuit, ST *)
FUNCTION_BLOCK Circuit
VAR_INPUT
(*-----команды и задания ручного режима----*)
	w_ManDevice	:DWORD; 	(*слово команд ручного режима контура *)

      (*общие*)
	Man_VE7     	: BOOL;     	(*VE7 Клапан промывки линии концентрата щелочи*)
	Man_P8      		: BOOL;		(*Р8 Насос-дозатор концентрата  кислоты*)
	Man_P9      		: BOOL;		(*Р9 Насос-дозатор концентрата  щелочи*)
	Man_P10     		: BOOL;		(*Р10 Насос-дозатор дезинфектанта*)

	ManSP_P1     	: REAL;
	ManSP_VR1    	: REAL;
(*----------------------------------------------*)
(*-----сигналы аварий для каждой операции мойки---------*)
	i_DiagSwillBackWater  		: BOOL;
	i_DiagSwillFreshWater 		: BOOL;
	i_DiagWashAlkaline 			: BOOL;
	i_DiagWashAcid 				: BOOL;
	i_DiagWashWater 			: BOOL;
	i_DiagThermDesinfection 		: BOOL;
	i_DiagChemicDesinfection 	: BOOL;
	i_DiagPrepareAlkaline 		: BOOL;
	i_DiagPrepareAcid 			: BOOL;
	i_DiagHandMode  			: BOOL;
	i_DiagDiagnostic  			: BOOL;

	i_Block_Q4_out  				: BOOL; 	(*блокировка выпуска для полоскания из Q4  - мин уровень и ph*)
	i_Block_Q4_in_level   		: BOOL; 	(*блокировка подачи в  Q4 по макс уровню*)
	i_Block_Q4_in_ph      		: BOOL; 	(*блокировка подачи в  Q4 по ph*)
	i_Ready_Route				: BOOL; 	(*сигнал о готовности выбранного маршрута, если 0 - запрет старта процесса или в паузу *)

	i_Block_SolPrep_Alk		: BOOL; 	(*блокировка подготовки раствора - идет мойка этим же р-ром по другому контуру*)
	i_Block_SolPrep_Acid	: BOOL; 	(*блокировка подготовки раствора - идет мойка этим же р-ром по другому контуру*)
	i_Block_Wash_Alk		: BOOL; 	(*блокировка мойки раствором - идет подготовка же р-ра по другому контуру*)
	i_Block_Wash_Acid		: BOOL; 	(*блокировка мойки раствором - идет подготовка же р-ра по другому контуру*)
	i_Alarm_LSmin_Alk		: BOOL;  	(*авария нижнего уровня в баке концентрата*)
	i_Alarm_LSmin_Acid		: BOOL; 	(*авария нижнего уровня в баке концентрата*)
	i_Alarm_LSmin_Dez 		: BOOL; 	(*авария нижнего уровня в баке концентрата*)
	i_Alarm_PE				: BOOL;		(*Превышение давления в контуре*)

	i_Pause                 		: BOOL;
	i_Stop                  		: BOOL; 	(*принудительная остановка процесса*)
	i_Start_AutoWashing     	: BOOL; 	(*старт мойки в автомате*)
	i_Start_HandMode        	: BOOL; 	(*старт ручного режима*)
	i_Start_PrepareAlkaline 	: BOOL; 	(*старт подготовки раствора щелочи*)
	i_Start_PrepareAcid     	: BOOL; 	(*старт подготовки раствора кислоты*)
	i_Start_Diagnostic      	: BOOL; 	(*старт диагностики клапанов*)
	i_ch_SwillBackWater     	: BOOL; 	(*выбор операции мойки*)
	i_ch_SwillFreshWater    	: BOOL; 	(*выбор операции мойки*)
	i_ch_WashAlkaline       	: BOOL; 	(*выбор операции мойки*)
	i_ch_WashWater1         	: BOOL; 	(*выбор операции мойки*)
	i_ch_WashAcid           	: BOOL; 	(*выбор операции мойки*)
	i_ch_WashWater2         	: BOOL; 	(*выбор операции мойки*)
	i_ch_ThermDesinfection  	: BOOL; 	(*выбор операции мойки*)
	i_ch_ChemicDesinfection : BOOL; 	(*выбор операции мойки*)

	i_FS1   			: BOOL;  (*имульсы расходомера дезинфектанта*)
	i_FC11  			: BOOL;  (*имульсы расходомера*)
	i_FS    			: BOOL;  (*датчик протока на возврате*)
	i_LSL   			: BOOL;  (*датчик уровня в циркуляционном баке*)
	i_LSM   			: BOOL;  (*датчик уровня в циркуляционном баке*)
	i_LSH   			: BOOL;  (*датчик уровня в циркуляционном баке*)

	i_TE1  			: REAL;  	(*температура на подаче*)
	i_TE2  			: REAL;      	(*температура на возврате*)
	i_TE_Q2			: REAL;    	(*температура в танке раствора щелочи*)
	i_LE_Q2			: REAL;    	(*уровень в танке раствора щелочи*)
	i_TE_Q3			: REAL;    	(*температура в танке раствора кислоты*)
	i_LE_Q3			: REAL;    	(*уровень в танке раствора кислоты*)
	i_QE   			: REAL;      	(*расчитанная концентрация % раствора*)
	i_QE_priv 		: REAL; 		(*приведенная проводимость к температуре*)

	i_TimeDelay      	: DINT ; 	(*время задержки вкл/выкл клапанов и насосов*)
	i_Time_LSH_on	: DINT ; 	(*время задержки срабатывания датчика верх уровня цирк бака*)
	i_Time_LSM_on	: DINT ; 	(*время задержки срабатывания датчика сред уровня цирк бака*)
	i_Time_LSM_off	: DINT ; 	(*время задержки отключения датчика сред уровня цирк бака*)
	i_Time_LSL_off 	: DINT ; 	(*время задержки отключения датчика ниж уровня цирк бака*)
	i_K_imp             	: REAL ;
	i_K_imp_dez    	: REAL ;

	i_AlkMixing        	: BOOL;          (*перемешивание щелочи*)
	i_AcidMixing      	: BOOL;          (*перемешивание кислоты*)

	i_TimeSwillBackWater  		: DINT ; 		(*время полоскания возвратной водой,с*)
	i_TimeSwillFreshWater 		: DINT ; 		(*время полоскания свежей водой,с*)
	i_TimeWashWater1      		: DINT ; 		(*время мойки 1 чистой водой,мин*)
	i_TimeSwillWashWater1 		: DINT ; 		(*время промывки водой со сбросом в Q4 после мойки 1 чистой водой,мин*)
	i_TempWashWater1      		: REAL ;		(*температруа мойки 1 чистой водой*)
	i_TimeWashWater2      		: DINT ; 		(*время мойки 2 чистой водой,мин*)
	i_TimeSwillWashWater2 		: DINT ; 		(*время промывки водой со сбросом в Q4 после мойки 2 чистой водой,мин*)
	i_TempWashWater2      		: REAL ;		(*температруа мойки 2 чистой водой*)
	i_TimeWashAlkaline    		: DINT ; 		(*время мойки щелочью,мин*)
	i_TempWashAlkaline    		: REAL ;		(*температура мойки щелочью*)
	i_TimeWashAcid        		: DINT ; 		(*время мойки кислотой,мин*)
	i_TempWashAcid        		: REAL ;		(*температура мойки кислотой*)
	i_TimeThermDesinf     		: DINT ; 		(*время термической дезинфекции,мин*)
	i_TempThermDesinf     		: REAL ; 	(*температура термической дезинфекции*)
	i_TempCoolThermDesinf 		: REAL ; 	(*температура охлаждения терм дезинфекции*)
	i_TimeChemicDesinf    		: DINT ; 		(*время химической дезинфекции,мин*)
	i_TimeSwillChemic       		: DINT ;  	(*время ополаскивания чистой водой после хим дехинфекции, если 0, то оставить дезинф в маршруте*)

	i_RouteType           			: DINT ; 		(*тип маршрута 1 - емкостной, 0 - замкнутый*)
	i_PumpCapacity        		: DINT ; 		(*производительность подающего насоса *)
	i_TimeDelayRetPump    		: DINT ; 		(*время задержки включения насоса возврата*)
	i_TimeDelayRetFlow    		: DINT ; 		(*время появления протока на возврате*)
	i_TimeAlarmBackFlow   		: DINT ; 		(*время аварии отсутствия обратного протока*)
	i_Numb_BackPump       		: DINT ; 		(*номер насоса возврата*)
	i_VolumeDesinf        			: DINT ; 		(*объем дезинфектанта*)
	i_Using_Q5          			: DINT;       	(*использование циркуляционного бака на мойках растворами и водой, 1 - использовать*)
	i_DeltaTempStartTime  		: DINT ; 		(*перепад температуры TE1-TE2 для начала терм дезинфекции*)

END_VAR
VAR_OUTPUT
(*---механизмы и устройства---*)
	w_qDevice	:DWORD; 	(*слово команд управления механизмами контура *)

	q_VE7 		: BOOL;		(*VE7 Клапан промывки линии концентрата щелочи*)
	q_P8  		: BOOL;		(*Р8 Насос-дозатор концентрата  кислоты*)
	q_P9 		: BOOL;		(*Р9 Насос-дозатор концентрата  щелочи*)
	q_P10  		: BOOL;		(*Р10 Насос-дозатор дезинфектанта*)

	q_Red  		: BOOL;		(*Светозвуковая сигнализация. Красный свет*)
	q_Yellow 	: BOOL;		(*Светозвуковая сигнализация. Желтый свет*)
	q_Green  	: BOOL;		(*Светозвуковая сигнализация. Зеленый свет*)
	q_Sirena	: BOOL;		(*Светозвуковая сигнализация. Зуммер*)



	q_AlarmBackFlow		:BOOL;  	(* авария протока на возврате*)
	q_Alarm_Empty_Q5		:BOOL;		(*авария опустошения цирк бака при работе на замкн маршруте*)
	q_Vis_tim_Process		:BOOL;
	q_Block_Solution_Alk		:BOOL;  	(*идет подготовка раствора - другим контурам не мыть*)
	q_Block_Solution_Acid	:BOOL; 		(*идет подготовка раствора - другим контурам не мыть*)
	q_Change_Mode 		:BOOL;		(*сигнал в ОР что режим не выбран*)
	q_Run_Process			:BOOL;  	(*в автоматическом режиме мойки идет подача моющих в маршрут - сигнал в маршрут*)
	q_End_AutoMode		:BOOL; 		(*закончен процесс мойки в автомате, импульс  - сигнал в маршрут*)

	q_SP_P1 				:REAL;		(*задание производительности на регулятор*)
	q_SP_VR1				:REAL;		(*задание температуры на регулятор*)
	q_VisuMode				:INT;		(*текущая стадия работы*)
	q_ModeQE 				:INT;     		(*режим выбора пересчета концентрации, 0-щелочь, 1-кислота*)
	q_Last_Time_min  		:DINT;  		(*расчет оставшихся минут процесса*)
	q_Last_Time_sec  		:DINT;  		(*расчет оставшихся секунд процесса*)
END_VAR

VAR
	Step                         		AT %M* : INT;
	Current_VolumeFC1  		AT %M*	: REAL;    (*текуший объем расходомера дезинфектанта*)
	Current_VolumeFC11 	AT %M*	: REAL;   (*текуший объем расходомера подачи*)

	FC1_start 				: BOOL;   	(*старт подсчета импульсов дезинф*)
	FC11_start				: BOOL;   	(*старт подсчета импульсов*)
	ZeroCount_FC1			: BOOL; 	(*обнуление счетчика дезинф*)
	ZeroCount_FC11			: BOOL; 	(*обнуление счетчика*)

  	fp_FC1_imp :R_TRIG ;  		(*определение переднего фронта импульса расходомера дезинфектанта*)
    	fp_FC11_imp:R_TRIG ;  		(*определение переднего фронта импульса расходомера подачи*)

	T_Control_TE :TON;    		(*таймер контроля набора температуры*)
	T_Control_QE :TON;   		(*таймер контроля набора концентрации*)
	T_Imp_EndAutoMode :TP; 	(*импульсный таймер выдачи сигнала "мойка закончена" в маршрут*)

	Preparation		:SolutionPrepar;
	Hand_Mode		:Manual;
	Diagn			:Diagnostic;
	Swill			:SwillWater;
	Wash_Solution	:WashSolution;
	Wash_Water		:WashWater;
	Chemical		:ChemicDesinf;
END_VAR
(*обнуление в начале скана*)
	w_qDevice := 0;

	q_VE7  := FALSE;
	q_P8 := FALSE;
	q_P9 := FALSE;
	q_P10 := FALSE;
	q_Red:=FALSE;
   	q_Green :=FALSE;
    	q_Yellow :=FALSE;
    	q_Sirena :=FALSE;

   	q_SP_P1 :=0.0 ;
    	q_SP_VR1 :=0.0 ;


    	q_AlarmBackFlow := FALSE;
    	q_Alarm_Empty_Q5:=FALSE;
    	q_Vis_tim_Process := FALSE;
    	q_Block_Solution_Alk:= FALSE;
    	q_Block_Solution_Acid:= FALSE;
    	q_Change_Mode:=FALSE;
    	q_Run_Process := FALSE;
    	q_End_AutoMode := FALSE;
    	q_VisuMode:=1;

    	T_Control_TE.IN:= FALSE;
    	T_Control_QE.IN:= FALSE;


 IF i_Stop THEN
     	Step:=0;
 END_IF;

CASE Step OF
0:(*контур выключен*)
   q_Change_Mode:=TRUE;

 IF i_Start_AutoWashing AND i_Ready_Route THEN  (*старт автомат режима при условии готовности маршрута*)
    Step:=1;
 ELSIF i_Start_HandMode THEN
    Hand_Mode.Step:=0;
    Step:=18;
 ELSIF i_Start_PrepareAlkaline AND NOT i_Block_SolPrep_Alk  THEN
    Preparation.Step:=0;
    Step:=19;
 ELSIF i_Start_PrepareAcid AND NOT i_Block_SolPrep_Acid THEN
    Preparation.Step:=0;
    Step:=20;
 ELSIF i_Start_Diagnostic  THEN
    Diagn.Step:=0;
    Step:=21;
 END_IF;

 T_Imp_EndAutoMode.IN := FALSE;


1: (*проверка на полоскание возвратной водой*)
 IF i_ch_SwillBackWater THEN
    Swill.Step:=0;
    Step:=2;
 ELSE
    Step:=3;
 END_IF;

2: (*полоскание возвратной водой*)

Swill(
	i_Diag:=i_DiagSwillBackWater ,
	i_Pause:=i_Pause ,
	i_fresh:=FALSE ,
	i_Block_Q4_out:=i_Block_Q4_out ,
	i_Block_Q4_in:=i_Block_Q4_in_level  ,
      i_Ready_Route := i_Ready_Route ,
	i_FS:=i_FS ,
	i_Current_VolumeFC11:=Current_VolumeFC11 ,
	i_TimeDelay:=i_TimeDelay ,
	i_TimeProcess:=i_TimeSwillBackWater ,
	i_RouteType:=i_RouteType ,
	i_PumpCapacity:=i_PumpCapacity ,
	i_TimeDelayRetPump:=i_TimeDelayRetPump ,
	i_TimeDelayRetFlow:=i_TimeDelayRetFlow ,
	i_TimeAlarmBackFlow:=i_TimeAlarmBackFlow ,
	q_VA541=>	w_qDevice.VA541 ,
	q_VA401=>	w_qDevice.VA401 ,
	q_VA201=>	w_qDevice.VA201 ,
	q_VA301=>	w_qDevice.VA301 ,
	q_VA41=>	w_qDevice.VA41 ,
	q_VA11=>	w_qDevice.VA11 ,
	q_VA21=>	w_qDevice.VA21 ,
	q_VA31=>	w_qDevice.VA31 ,
	q_VA551=>	w_qDevice.VA5 ,
	q_VA501=>	w_qDevice.VA501 ,
	q_VA51=>	w_qDevice.VA51 ,
	q_VA511=>	w_qDevice.VA511 ,
	q_VA521=>	w_qDevice.VA521 ,
	q_VA531=>	w_qDevice.VA531 ,
	q_P1=>		w_qDevice.P1 ,
	q_Red=>q_Red ,
	q_Yellow=>q_Yellow ,
	q_Green=>q_Green ,
	q_Sirena=>q_Sirena ,
	q_BackPump=>		w_qDevice.BackPump ,
	q_Heating_VR1=>	w_qDevice.Heating_VR1 ,
	q_AlarmBackFlow=>q_AlarmBackFlow ,
	q_Vis_tim_Process=>q_Vis_tim_Process ,
	q_FC11_start=>FC11_start ,
	q_ZeroCount_FC11=>ZeroCount_FC11 ,
	q_SP_P1=>q_SP_P1 ,
	q_SP_VR1=>q_SP_VR1 ,
	q_VisuMode=>q_VisuMode );
  q_Last_Time_min:=Swill.Last_Time_min;
  q_Last_Time_sec:=Swill.Last_Time_sec;
 q_Run_Process := (Swill.Step< 4); (*идет подача моющих в маршрут - сигнал в маршрут*)

  IF Swill.Step=4 THEN
     Step:=3;
  END_IF;


3: (*проверка на полоскание свежей водой*)
 IF i_ch_SwillFreshWater THEN
    Swill.Step:=0;
    Step:=4;
 ELSE
    Step:=5;
 END_IF;

4: (*полоскание свежей водой*)

Swill(
	i_Diag:=i_DiagSwillFreshWater ,
	i_Pause:=i_Pause ,
	i_fresh:=TRUE ,
	i_Block_Q4_out:=i_Block_Q4_out ,
	i_Block_Q4_in:=i_Block_Q4_in_level ,
      i_Ready_Route := i_Ready_Route ,
	i_FS:=i_FS ,
	i_Current_VolumeFC11:=Current_VolumeFC11 ,
	i_TimeDelay:=i_TimeDelay ,
	i_TimeProcess:=i_TimeSwillFreshWater ,
	i_RouteType:=i_RouteType ,
	i_PumpCapacity:=i_PumpCapacity ,
	i_TimeDelayRetPump:=i_TimeDelayRetPump ,
	i_TimeDelayRetFlow:=i_TimeDelayRetFlow ,
	i_TimeAlarmBackFlow:=i_TimeAlarmBackFlow ,
	q_VA541=>	w_qDevice.VA541 ,
	q_VA401=>	w_qDevice.VA401 ,
	q_VA201=>	w_qDevice.VA201 ,
	q_VA301=>	w_qDevice.VA301 ,
	q_VA41=>	w_qDevice.VA41 ,
	q_VA11=>	w_qDevice.VA11 ,
	q_VA21=>	w_qDevice.VA21 ,
	q_VA31=>	w_qDevice.VA31 ,
	q_VA551=>	w_qDevice.VA5 ,
	q_VA501=>	w_qDevice.VA501 ,
	q_VA51=>	w_qDevice.VA51 ,
	q_VA511=>	w_qDevice.VA511 ,
	q_VA521=>	w_qDevice.VA521 ,
	q_VA531=>	w_qDevice.VA531 ,
	q_P1=>		w_qDevice.P1 ,
	q_Red=>q_Red ,
	q_Yellow=>q_Yellow ,
	q_Green=>q_Green ,
	q_Sirena=>q_Sirena ,
	q_BackPump=>	w_qDevice.BackPump ,
	q_Heating_VR1=>	w_qDevice.Heating_VR1 ,
	q_AlarmBackFlow=>q_AlarmBackFlow ,
	q_Vis_tim_Process=>q_Vis_tim_Process ,
	q_FC11_start=>FC11_start ,
	q_ZeroCount_FC11=>ZeroCount_FC11 ,
	q_SP_P1=>q_SP_P1 ,
	q_SP_VR1=>q_SP_VR1 ,
	q_VisuMode=>q_VisuMode );
  q_Last_Time_min:=Swill.Last_Time_min;
  q_Last_Time_sec:=Swill.Last_Time_sec;
  q_Run_Process := (Swill.Step< 4); (*идет подача моющих в маршрут - сигнал в маршрут*)

  IF Swill.Step=4 THEN
     Step:=5;
  END_IF;


5: (*проверка на мойку щелочью*)
  IF i_ch_WashAlkaline THEN
       IF NOT i_Block_Wash_Alk THEN (*если не идет подготовка р-ра по другому контуру*)
           Wash_Solution.Step:=0;
           Step:=6;
       ELSE
           q_VisuMode:=17;
       END_IF;
  ELSE
    Step:=7;
  END_IF;


6: (*мойка щелочью*)
    q_ModeQE:=0;  (*режим выбора пересчета концентрации*)
Wash_Solution(
	i_Diag:=i_DiagWashAlkaline ,
	i_Diag_Preparation:=i_DiagPrepareAlkaline,
	i_Pause:=i_Pause ,
	i_Block_Q4_out:=i_Block_Q4_out ,
	i_Block_Q4_in:=i_Block_Q4_in_level AND i_Block_Q4_in_ph  ,
	i_Block_SolPrep:=i_Block_SolPrep_Alk ,
	i_Alarm_LSmin:=i_Alarm_LSmin_Alk ,
      i_Ready_Route := i_Ready_Route ,
      i_Alk:=TRUE,
	i_FS:=i_FS ,
	i_LSL:=i_LSL ,
	i_LSM:=i_LSM ,
	i_LSH:=i_LSH ,
	i_Mixing:=i_AlkMixing ,
	i_TE1:=i_TE1 ,
	i_TE2:=i_TE2 ,
	i_TE_tank:=i_TE_Q2 ,
	i_LE_tank:=i_LE_Q2 ,
	i_QE:=i_QE ,
	i_QE_priv:=i_QE_priv ,
	i_Current_VolumeFC11:=Current_VolumeFC11 ,
	i_MaxCondPrep:=MaxCondPrepAlk ,
	i_MinCondPrep:=MinCondPrepAlk ,
	i_MaxTempPrep:=MaxTempPrepAlk ,
	i_MinTempPrep:=MinTempPrepAlk ,
	i_LvlPrep:=LvlPrepAlk ,
	Cond_Q4:=CondAlk_Q4 ,
	i_TimeDelay:=i_TimeDelay ,
	i_Time_LSH_on:=i_Time_LSH_on ,
	i_Time_LSM_on:=i_Time_LSM_on ,
	i_Time_LSM_off:=i_Time_LSM_off ,
	i_Time_LSL_off:=i_Time_LSL_off ,
	i_TimeProcess:=i_TimeWashAlkaline ,
	i_TempProcess:=i_TempWashAlkaline ,
	i_RouteType:=i_RouteType ,
	i_PumpCapacity:=i_PumpCapacity ,
	i_TimeDelayRetPump:=i_TimeDelayRetPump ,
	i_TimeDelayRetFlow:=i_TimeDelayRetFlow ,
	i_TimeAlarmBackFlow:=i_TimeAlarmBackFlow ,
       i_Using_Q5 := i_Using_Q5 ,
	q_VA541=>	w_qDevice.VA541 ,
	q_VA401=>	w_qDevice.VA401 ,
	q_VA201=>	w_qDevice.VA201 ,
	q_VA41=>	w_qDevice.VA41 ,
	q_VA11=>	w_qDevice.VA11 ,
	q_VA21=>	w_qDevice.VA21 ,
	q_VA551=>	w_qDevice.VA5 ,
	q_VA501=>	w_qDevice.VA501 ,
	q_VA51=>	w_qDevice.VA51 ,
	q_VA511=>	w_qDevice.VA511 ,
	q_VA521=>	w_qDevice.VA521 ,
	q_VA531=>	w_qDevice.VA531 ,
	q_VE11=>	q_VE7 ,
	q_P1=>		w_qDevice.P1 ,
	q_P10=>q_P9 ,
	q_Red=>q_Red ,
	q_Yellow=>q_Yellow ,
	q_Green=>q_Green ,
	q_Sirena=>q_Sirena ,
	q_BackPump=>	w_qDevice.BackPump ,
	q_Heating_VR1=>w_qDevice.Heating_VR1 ,
	q_AlarmBackFlow=>q_AlarmBackFlow ,
    q_Alarm_Empty_Q5=>q_Alarm_Empty_Q5 ,
	q_Vis_tim_Process=>q_Vis_tim_Process ,
	q_FC11_start=>FC11_start ,
	q_ZeroCount_FC11=>ZeroCount_FC11 ,
	q_Block_Solution=>q_Block_Solution_Alk ,
	q_SP_P1=>q_SP_P1 ,
	q_SP_VR1=>q_SP_VR1 ,
	q_VisuMode=>q_VisuMode );
  q_Last_Time_min:=Wash_Solution.Last_Time_min;
  q_Last_Time_sec:=Wash_Solution.Last_Time_sec;

 T_Control_TE.IN:=w_qDevice.Heating_VR1 AND (i_TE1<(q_SP_VR1-2.0));
 T_Control_QE.IN:=Wash_Solution.q_P10;
 q_Run_Process := (Wash_Solution.Step>4) AND (Wash_Solution.Step< 19); (*идет подача моющих в маршрут - сигнал в маршрут*)

  IF Wash_Solution.Step=19 THEN
     Step:=7;
  END_IF;

7: (*проверка на мойку чистой водой 1 после щелочи*)
 IF i_ch_WashWater1 THEN
    Wash_Water.Step:=0;
    Step:=8;
 ELSE
    Step:=9;
 END_IF;

8: (*мойка чистой водой 1 после щелочи*)
Wash_Water(
	i_Diag:=i_DiagWashWater ,
	i_Pause:=i_Pause ,
	i_Block_Q4_out:=i_Block_Q4_out ,
	i_Block_Q4_in:=i_Block_Q4_in_level ,
      i_Ready_Route := i_Ready_Route ,
	i_type:=0 ,
	i_FS:=i_FS ,
	i_LSL:=i_LSL ,
	i_LSM:=i_LSM ,
	i_LSH:=i_LSH ,
	i_TE1:=i_TE1 ,
	i_TE2:=i_TE2 ,
	i_Current_VolumeFC1:=Current_VolumeFC1 ,
	i_Current_VolumeFC11:=Current_VolumeFC11 ,
	i_TimeDelay:=i_TimeDelay ,
	i_Time_LSH_on:=i_Time_LSH_on ,
	i_Time_LSM_on:=i_Time_LSM_on ,
	i_Time_LSM_off:=i_Time_LSM_off ,
	i_Time_LSL_off:=i_Time_LSL_off ,
	i_TimeProcess:=i_TimeWashWater1 ,
       i_TimeSwillWater:=i_TimeSwillWashWater1 ,
	i_TempProcess:=i_TempWashWater1 ,
	i_DeltaTempStartTime:=i_DeltaTempStartTime ,
	i_TempCool:=i_TempCoolThermDesinf ,
	i_RouteType:=i_RouteType ,
	i_PumpCapacity:=i_PumpCapacity ,
	i_TimeDelayRetPump:=i_TimeDelayRetPump ,
	i_TimeDelayRetFlow:=i_TimeDelayRetFlow ,
	i_TimeAlarmBackFlow:=i_TimeAlarmBackFlow ,
       i_Using_Q5 := i_Using_Q5 ,
	i_VolumeDesinf:=i_VolumeDesinf ,
	q_VA541=>	w_qDevice.VA541 ,
	q_VA401=>	w_qDevice.VA401 ,
	q_VA11=>	w_qDevice.VA11 ,
	q_VA551=>	w_qDevice.VA5 ,
	q_VA501=>	w_qDevice.VA501 ,
	q_VA51=>	w_qDevice.VA51 ,
	q_VA511=>	w_qDevice.VA511 ,
	q_VA521=>	w_qDevice.VA521 ,
	q_VA531=>	w_qDevice.VA531 ,
	q_VE551=>	w_qDevice.VE551 ,
	q_P1=>		w_qDevice.P1 ,
	q_P12=>q_P10 ,
	q_Red=>q_Red ,
	q_Yellow=>q_Yellow ,
	q_Green=>q_Green ,
	q_Sirena=>q_Sirena ,
	q_BackPump=>	w_qDevice.BackPump ,
	q_Heating_VR1=>w_qDevice.Heating_VR1 ,
	q_AlarmBackFlow=>q_AlarmBackFlow ,
    q_Alarm_Empty_Q5=>q_Alarm_Empty_Q5 ,
	q_Vis_tim_Process=>q_Vis_tim_Process ,
	q_FC1_start=>FC1_start ,
	q_FC11_start=>FC11_start ,
	q_ZeroCount_FC1=>ZeroCount_FC1 ,
	q_ZeroCount_FC11=>ZeroCount_FC11 ,
	q_SP_P1=>q_SP_P1 ,
	q_SP_VR1=>q_SP_VR1 ,
	q_VisuMode=>q_VisuMode );
  q_Last_Time_min:=Wash_Water.Last_Time_min;
  q_Last_Time_sec:=Wash_Water.Last_Time_sec;

 T_Control_TE.IN:=w_qDevice.Heating_VR1 AND (i_TE1<(q_SP_VR1-2.0));
 q_Run_Process := (Wash_Water.Step<10); (*идет подача моющих в маршрут - сигнал в маршрут*)

  IF Wash_Water.Step=10 THEN
     Step:=9;
  END_IF;


9: (*проверка на мойку кислотой*)
  IF i_ch_WashAcid THEN
       IF NOT i_Block_Wash_Acid THEN (*если не идет подготовка р-ра по другому контуру*)
           Wash_Solution.Step:=0;
           Step:=10;
       ELSE
           q_VisuMode:=17;
       END_IF;
  ELSE
    Step:=11;
  END_IF;

10: (*мойка кислотой*)
    q_ModeQE:=1;  (*режим выбора пересчета концентрации*)
Wash_Solution(
	i_Diag:=i_DiagWashAcid ,
	i_Diag_Preparation:=i_DiagPrepareAlkaline,
	i_Pause:=i_Pause ,
	i_Block_Q4_out:=i_Block_Q4_out ,
	i_Block_Q4_in:=i_Block_Q4_in_level AND i_Block_Q4_in_ph  ,
	i_Block_SolPrep:=i_Block_SolPrep_Acid ,
	i_Alarm_LSmin:=i_Alarm_LSmin_Acid ,
      i_Ready_Route := i_Ready_Route ,
      i_Alk:=FALSE,
	i_FS:=i_FS ,
	i_LSL:=i_LSL ,
	i_LSM:=i_LSM ,
	i_LSH:=i_LSH ,
	i_Mixing:=i_AcidMixing ,
	i_TE1:=i_TE1 ,
	i_TE2:=i_TE2 ,
	i_TE_tank:=i_TE_Q3 ,
	i_LE_tank:=i_LE_Q3 ,
	i_QE:=i_QE ,
	i_QE_priv:=i_QE_priv ,
	i_Current_VolumeFC11:=Current_VolumeFC11 ,
	i_MaxCondPrep:=MaxCondPrepAcid ,
	i_MinCondPrep:=MinCondPrepAcid ,
	i_MaxTempPrep:=MaxTempPrepAcid ,
	i_MinTempPrep:=MinTempPrepAcid ,
	i_LvlPrep:=LvlPrepAcid ,
	Cond_Q4:=CondAcid_Q4 ,
	i_TimeDelay:=i_TimeDelay ,
	i_Time_LSH_on:=i_Time_LSH_on ,
	i_Time_LSM_on:=i_Time_LSM_on ,
	i_Time_LSM_off:=i_Time_LSM_off ,
	i_Time_LSL_off:=i_Time_LSL_off ,
	i_TimeProcess:=i_TimeWashAcid,
	i_TempProcess:=i_TempWashAcid ,
	i_RouteType:=i_RouteType ,
	i_PumpCapacity:=i_PumpCapacity ,
	i_TimeDelayRetPump:=i_TimeDelayRetPump ,
	i_TimeDelayRetFlow:=i_TimeDelayRetFlow ,
	i_TimeAlarmBackFlow:=i_TimeAlarmBackFlow ,
       i_Using_Q5 := i_Using_Q5 ,
	q_VA541=>	w_qDevice.VA541 ,
	q_VA401=>	w_qDevice.VA401 ,
	q_VA201=>	w_qDevice.VA301 ,
	q_VA41=>	w_qDevice.VA41 ,
	q_VA11=>	w_qDevice.VA11 ,
	q_VA21=>	w_qDevice.VA31 ,
	q_VA551=>	w_qDevice.VA5 ,
	q_VA501=>	w_qDevice.VA501 ,
	q_VA51=>	w_qDevice.VA51 ,
	q_VA511=>	w_qDevice.VA511 ,
	q_VA521=>	w_qDevice.VA521 ,
	q_VA531=>	w_qDevice.VA531 ,
	q_VE11=> ,
	q_P1=>		w_qDevice.P1 ,
	q_P10=>q_P8 ,
	q_Red=>q_Red ,
	q_Yellow=>q_Yellow ,
	q_Green=>q_Green ,
	q_Sirena=>q_Sirena ,
	q_BackPump=>		w_qDevice.BackPump ,
	q_Heating_VR1=>	w_qDevice.Heating_VR1 ,
	q_AlarmBackFlow=>q_AlarmBackFlow ,
    q_Alarm_Empty_Q5=>q_Alarm_Empty_Q5 ,
	q_Vis_tim_Process=>q_Vis_tim_Process ,
	q_FC11_start=>FC11_start ,
	q_ZeroCount_FC11=>ZeroCount_FC11 ,
	q_Block_Solution=>q_Block_Solution_Acid ,
	q_SP_P1=>q_SP_P1 ,
	q_SP_VR1=>q_SP_VR1 ,
	q_VisuMode=>q_VisuMode );
  q_Last_Time_min:=Wash_Solution.Last_Time_min;
  q_Last_Time_sec:=Wash_Solution.Last_Time_sec;

 T_Control_TE.IN:=w_qDevice.Heating_VR1 AND (i_TE1<(q_SP_VR1-2.0));
 T_Control_QE.IN:=Wash_Solution.q_P10;
 q_Run_Process := (Wash_Solution.Step>4) AND (Wash_Solution.Step< 19); (*идет подача моющих в маршрут - сигнал в маршрут*)

  IF Wash_Solution.Step=19 THEN
     Step:=11;
  END_IF;

11: (*проверка на мойку чистой водой 2 после кислоты*)
 IF i_ch_WashWater2 THEN
    Wash_Water.Step:=0;
    Step:=12;
 ELSE
    Step:=13;
 END_IF;

12: (*мойка чистой водой 2 после кислоты*)
Wash_Water(
	i_Diag:=i_DiagWashWater ,
	i_Pause:=i_Pause ,
	i_Block_Q4_out:=i_Block_Q4_out ,
	i_Block_Q4_in:=i_Block_Q4_in_level ,
      i_Ready_Route := i_Ready_Route ,
	i_type:=0 ,
	i_FS:=i_FS ,
	i_LSL:=i_LSL ,
	i_LSM:=i_LSM ,
	i_LSH:=i_LSH ,
	i_TE1:=i_TE1 ,
	i_TE2:=i_TE2 ,
	i_Current_VolumeFC1:=Current_VolumeFC1 ,
	i_Current_VolumeFC11:=Current_VolumeFC11 ,
	i_TimeDelay:=i_TimeDelay ,
	i_Time_LSH_on:=i_Time_LSH_on ,
	i_Time_LSM_on:=i_Time_LSM_on ,
	i_Time_LSM_off:=i_Time_LSM_off ,
	i_Time_LSL_off:=i_Time_LSL_off ,
	i_TimeProcess:=i_TimeWashWater2 ,
       i_TimeSwillWater:=i_TimeSwillWashWater2 ,
	i_TempProcess:=i_TempWashWater2 ,
	i_DeltaTempStartTime:=i_DeltaTempStartTime ,
	i_TempCool:=i_TempCoolThermDesinf ,
	i_RouteType:=i_RouteType ,
	i_PumpCapacity:=i_PumpCapacity ,
	i_TimeDelayRetPump:=i_TimeDelayRetPump ,
	i_TimeDelayRetFlow:=i_TimeDelayRetFlow ,
	i_TimeAlarmBackFlow:=i_TimeAlarmBackFlow ,
       i_Using_Q5 := i_Using_Q5 ,
	i_VolumeDesinf:=i_VolumeDesinf ,
	q_VA541=>	w_qDevice.VA541 ,
	q_VA401=>	w_qDevice.VA401 ,
	q_VA11=>	w_qDevice.VA11 ,
	q_VA551=>	w_qDevice.VA5 ,
	q_VA501=>	w_qDevice.VA501 ,
	q_VA51=>	w_qDevice.VA51 ,
	q_VA511=>	w_qDevice.VA511 ,
	q_VA521=>	w_qDevice.VA521 ,
	q_VA531=>	w_qDevice.VA531 ,
	q_VE551=>	w_qDevice.VE551 ,
	q_P1=>		w_qDevice.P1 ,
	q_P12=>q_P10 ,
	q_Red=>q_Red ,
	q_Yellow=>q_Yellow ,
	q_Green=>q_Green ,
	q_Sirena=>q_Sirena ,
	q_BackPump=>	w_qDevice.BackPump ,
	q_Heating_VR1=>	w_qDevice.Heating_VR1 ,
	q_AlarmBackFlow=>q_AlarmBackFlow ,
    q_Alarm_Empty_Q5=>q_Alarm_Empty_Q5 ,
	q_Vis_tim_Process=>q_Vis_tim_Process ,
	q_FC1_start=>FC1_start ,
	q_FC11_start=>FC11_start ,
	q_ZeroCount_FC1=>ZeroCount_FC1 ,
	q_ZeroCount_FC11=>ZeroCount_FC11 ,
	q_SP_P1=>q_SP_P1 ,
	q_SP_VR1=>q_SP_VR1 ,
	q_VisuMode=>q_VisuMode );
  q_Last_Time_min:=Wash_Water.Last_Time_min;
  q_Last_Time_sec:=Wash_Water.Last_Time_sec;

 T_Control_TE.IN:=w_qDevice.Heating_VR1 AND (i_TE1<(q_SP_VR1-2.0));
 q_Run_Process := (Wash_Water.Step<10); (*идет подача моющих в маршрут - сигнал в маршрут*)

  IF Wash_Water.Step=10 THEN
     Step:=13;
  END_IF;

13: (*проверка на химическую дезинфекцию*)
 IF i_ch_ChemicDesinfection THEN
    Chemical.Step:=0;
    Step:=14;
 ELSE
    Step:=15;
 END_IF;

